FUNCTION_BLOCK "FB24 - Gestione Mov Assi"	// FB 24
TITLE = GESTIONE ASSI STAZIONE OP60
VERSION : 0.1
VAR_INPUT
  INDIRIZZO_INIZIALE_E_A : DINT ;	//INDIRIZZO INIZIALE I/O (VEDI CONFIGURAZIONE HARDWARE)
  OK_FOR_COMMANDS : BOOL ;	//TUTTO PRONTO PER I COMANDI
  RESET_ALLARMI : BOOL ;	//1=RESET ALLARMI AZIONAMENTO
  STOP : BOOL ;	//0=STOP DI TUTTI I MOVIMENTI
  TARGET_POSIZIONE : DINT ;	//TARGET DI POSIZIONAMENTO ASSOLUTO
  TARGET_INCREMENTALE : DINT ;	//SPOSTAMENTO IN MODO INCREMENTALE
  OVERRIDE : INT ;	//OVVERIDE DI VELOCITA'
  JOG_PIU : BOOL ;	//COMANDO JOG PIU'
  JOG_MENO : BOOL ;	//COMANDO JOG MENO
  IN_PKE : WORD ;
  IN_IND : WORD ;
  IN_PWE : DINT ;
  ASSE_SU_HOME : BOOL ;	//ASSE GIA' SU POSIZIONE DI HOME
END_VAR
VAR_OUTPUT
  OUT_PKE : WORD ;
  OUT_IND : WORD ;
  OUT_PWE : DINT ;
  POSIZIONE_ATTUALE : DINT ;
  POSIZIONE_RAGGIUNTA : BOOL ;	//POSIZIONAMENTO ULTIMATO
  HOME_OK : BOOL ;	//1=ASSE RIFERITO
  RIPOSIZIONAMENTO_OK : BOOL ;	//1=RIPOSIZIONAMENTO EFFETTUATO
  ASSE_FERMO_NO_JOB : BOOL ;	//1=ASSE FERMO E NESSUN JOB IN CORSO
  AZIONAMENTO_OK : BOOL ;	//1=AZIONAMENTO PRONTO
  AZIONAMENTO_FAULT : BOOL ;	//1=AZIONAMENTO IN ALLARME
  CAMMA_DI_RIFERIMENTO : BOOL ;	//1=ASSE SU CAMMA DI RIFERIMENTO
  OLTRECORSA_NEGATIVO : BOOL ;	//1=ASSE SU OLTRECORSA HARDWARE NEGATIVO
  OLTRECORSA_POSITIVO : BOOL ;	//1=ASSE SU OLTRECORSA HARDWARE POSITIVO
  FINECORSA_SOFTWARE_NEG : BOOL ;	//1=FINECORSA SOFTWARE NEGATIVO
  FINECORSA_SOFTWARE_POS : BOOL ;	//1=FINECORSA SOFTWARE POSITIVO
  FRENO : BOOL ;	//1=APRIRE IL FRENO DI STAZIONAMENTO
END_VAR
VAR_IN_OUT
  START_ASSOLUTO : BOOL ;	//1=START POSIZIONAMENTO ASSOLUTO
  START_INCREMENTALE : BOOL ;	//1=START POSIZIONAMENTO INCREMENTALE
  START_HOME : BOOL ;	//1=START RICERCA ZERO
  START_RIPOSIZIONAMENTO : BOOL ;	//1=START POSIZIONAMENTO SU POSIZIONE INIZIALE
END_VAR
VAR
  SCELTA_BLOCCO : WORD ;
  BLOCCO_ATTUALE : WORD ;
  INVIA_JOB1 : BOOL ;	//INVIO COMANDO DI CARICA BLOCCO ASSOLUTO
  JOB1_ULTIMATO : BOOL ;	//IL NUOVO BLOCCO DI MOVIMENTO ASSOLUTO E' STATO INVIATO
  INVIA_JOB2 : BOOL ;	//INVIO COMANDO DI CARICA BLOCCO INCREMENTALE
  JOB2_ULTIMATO : BOOL ;	//IL NUOVO BLOCCO DI MOVIMENTO INCREMENTALE E' STATO INVIATO
  GIA_IN_POSIZIONE : BOOL ;	//POSIZIONAMENTO NON NECESSARIO PER ASSE GIA' IN POSIZIONE
  PACO1 : STRUCT
   PACO1_8 : BOOL ;	//1=MARCIA A IMPULSI 1
   PACO1_9 : BOOL ;	//1=MARCIA 1 IMPULSI 2
   PACO1_10 : BOOL ;	//1=ABILITA IL COMANDO (DA METTERE A 1 QUANDO PAST1.9=1)
   PACO1_11 : BOOL ;	//1=AVVIA IL RIFERIMENTO DELL'ASSE
   PACO1_12 : BOOL ;	//RISERVATO
   PACO1_13 : BOOL ;	//1=CAMBIO BLOCCO ESTERNO
   PACO1_14 : BOOL ;	//RISERVATO
   PACO1_15 : BOOL ;	//RISERVATO
   PACO1_0 : BOOL ;	//1=INSERITO 0=DISINSERITO
   PACO1_1 : BOOL ;	//1=INSERITO 0=DISINSERITO
   PACO1_2 : BOOL ;	//1=INSERITO 0=DISINSERITO
   PACO1_3 : BOOL ;	//0=BLOCCO IMPULSI (IL MOTORE SI FERMA PER INERZIA)
   PACO1_4 : BOOL ;	//1=OK 0=STOP ASSE E CANCELLAZIONE PERCORSO RESISDUO
   PACO1_5 : BOOL ;	//1=OK 0=STOP ASSE E ULTIMAZIONE MOVIMENTO CON FRONTE 0-->1
   PACO1_6 : BOOL ;	//0-->1=ATTIVARE L'ORDINE DI SPOSTAMENTO
   PACO1_7 : BOOL ;	//1=TACITAZIONE ALLARME
  END_STRUCT ;
  PAST1 : STRUCT
   PAST1_8 : BOOL ;	//1=NESSUN ERRORE D'INSEGUIMENTO
   PAST1_9 : BOOL ;	//1=SLAVE OK E PRONTO A RICEVERE COMANDI
   PAST1_10 : BOOL ;	//1=POSIZIONE RAGGIUNTA
   PAST1_11 : BOOL ;	//1=ASSE RIFERITO
   PAST1_12 : BOOL ;	//1=POSIZIONAMENTO IN CORSO
   PAST1_13 : BOOL ;	//1=MOTORE FERMO
   PAST1_14 : BOOL ;	//RISERVATO
   PAST1_15 : BOOL ;	//RISERVATO
   PAST1_0 : BOOL ;	//1=PRONTO ALL'INSERZIONE
   PAST1_1 : BOOL ;	//1=PRONTO AL FUNZIONAMENTO
   PAST1_2 : BOOL ;	//STATO ABILITAZIONE REGOLATORE
   PAST1_3 : BOOL ;	//1=PRESEZA GUASTI
   PAST1_4 : BOOL ;	//1=DISINSERIMENTO 2 ASSENTE
   PAST1_5 : BOOL ;	//1=DISINSERIMENTO 3 ASSENTE
   PAST1_6 : BOOL ;	//1=BLOCCO ALL'INSERZIONE
   PAST1_7 : BOOL ;	//1=PRESENZA AVVISI
  END_STRUCT ;
  DIGin : STRUCT
   DIGin_8 : BOOL ;
   DIGin_9 : BOOL ;
   DIGin_10 : BOOL ;
   DIGin_11 : BOOL ;
   DIGin_12 : BOOL ;
   DIGin_13 : BOOL ;
   DIGin_14 : BOOL ;
   DIGin_15 : BOOL ;
   DIGin_0 : BOOL ;	//1=ASSE SU CAMMA DI HOME
   DIGin_1 : BOOL ;	//1=ASSE SU EXTRACORSA NEGATIVO
   DIGin_2 : BOOL ;	//1=ASSE SU EXTRACORSA POSITIVO
   DIGin_3 : BOOL ;
   DIGin_4 : BOOL ;
   DIGin_5 : BOOL ;
   DIGin_6 : BOOL ;
   DIGin_7 : BOOL ;
  END_STRUCT ;
  AUX1 : BOOL ;	//APPOGGIO PER FRONTE
  AUX2 : BOOL ;	//APPOGGIO PER FRONTE
  AUX3 : BOOL ;	//APPOGGIO PER FRONTE
  AUX4 : BOOL ;	//APPOGGIO PER FRONTE
  AUX5 : BOOL ;	//APPOGGIO PER FRONTE
  AUX6 : BOOL ;	//APPOGGIO PER FRONTE
  AUX7 : BOOL ;	//APPOGGIO PER FRONTE
  VERIFICA_SPOSTAMENTO : DINT ;	//DIFFERENZA TRA TARGET E POSIZIONE ATTUALE
  PAST2 : STRUCT
   PAST2_8 : BOOL ;	//1=TACITARE IL GUASTO 608
   PAST2_9 : BOOL ;	//1=ATTUALE MOTORE 1.SEGNALE
   PAST2_10 : BOOL ;	//1=ATTUALE MOTORE 2.SEGNALE
   PAST2_11 : BOOL ;	//1=RISERVATO
   PAST2_12 : BOOL ;
   PAST2_13 : BOOL ;
   PAST2_14 : BOOL ;
   PAST2_15 : BOOL ;
   PAST2_0 : BOOL ;
   PAST2_1 : BOOL ;
   PAST2_2 : BOOL ;
   PAST2_3 : BOOL ;	//PRIMO FILTRO DEL RIFERIMENTO ATTIVO
   PAST2_4 : BOOL ;	//BLOCCO DELL'INTEGRATORE NEL REGOLATORE DI VELOCITA'
   PAST2_5 : BOOL ;	//APRIRE IL FRENO DI STAZIONAMENTO
   PAST2_6 : BOOL ;	//BLOCCO DELL'INTEGRATORE NEL REGOLATORE DI VELOCITA'
   PAST2_7 : BOOL ;	//SCELTO L'ASSE IN PARCHEGGIO
  END_STRUCT ;
  POS_PAST : STRUCT
   POS_PAST_0 : BOOL ;	//FUNZIONAMENTO A SEGUIRE
   POS_PAST_1 : BOOL ;	//LIMITAZIONE DELLA VELOCITA' LINEARE ATTIVA
   POS_PAST_2 : BOOL ;	//C'E' IL RIFERIMENTO
   POS_PAST_3 : BOOL ;	//BIT DI FUNZIONE
   POS_PAST_4 : BOOL ;	//L'ASSE SI SPOSTA IN AVANTI
   POS_PAST_5 : BOOL ;	//L'ASSE SI SPOSTA INDIETRO
   POS_PAST_6 : BOOL ;	//FINECORSA SOFTWARE MENO
   POS_PAST_7 : BOOL ;	//FINECORSA SOFTWARE PIU'
   POS_PAST_8 : BOOL ;	//SEGNALE D'INSERZIONE DELLA CAMMA 1
   POS_PAST_9 : BOOL ;	//SEGNALE D'INSERZIONE DELLA CAMMA 2
   POS_PAST_10 : BOOL ;	//USCITA DIRETTA 1 CON IL BLOCCO DI SPOSTAMENTO
   POS_PAST_11 : BOOL ;	//USCITA DIRETTA 2 CON IL BLOCCO DI SPOSTAMENTO
   POS_PAST_12 : BOOL ;	//RISERVATO
   POS_PAST_13 : BOOL ;	//RISERVATO
   POS_PAST_14 : BOOL ;	//RISERVATO
   POS_PAST_15 : BOOL ;	//RISERVATO
  END_STRUCT ;
END_VAR
BEGIN
NETWORK
TITLE = AGGIORNAMENTO IMMAGINE INGRESSI
      L     #INDIRIZZO_INIZIALE_E_A;
      L     8;
      +I;
      SLD   3;
      T     MD 100;
      L     PIW [MD 100];	//;PAST1
      T     DIW 52;
      L     MD 100;
      SRW   3;
      L     2;
      +D;
      SLW   3;
      T     MD 100;
//;
      L     PIW [MD 100];	//;BLOCCO ATTUALE
      T     #BLOCCO_ATTUALE;
      L     MD 100;
      SRW   3;
      L     2;
      +D;
      SLW   3;
      T     MD 100;
//;
      L     PIW [MD 100];	//;POS PAST
      T     DIW 64;
      L     MD 100;
      SRW   3;
      L     2;
      +D;
      SLW   3;
      T     MD 100;
//;
      L     PIW [MD 100];	//;PAST 2
      T     DIW 62;
      L     MD 100;
      SRW   3;
      L     2;
      +D;
      SLW   3;
      T     MD 100;
//;
      L     PID [MD 100];	//; POSIZIONE ATTUALE
      T     #POSIZIONE_ATTUALE;
      L     MD 100;
      SRW   3;
      L     4;
      +D;
      SLW   3;
      T     MD 100;
//;
      L     PIW [MD 100];	//;INGRESSI DIGITALI
      T     DIW 54;
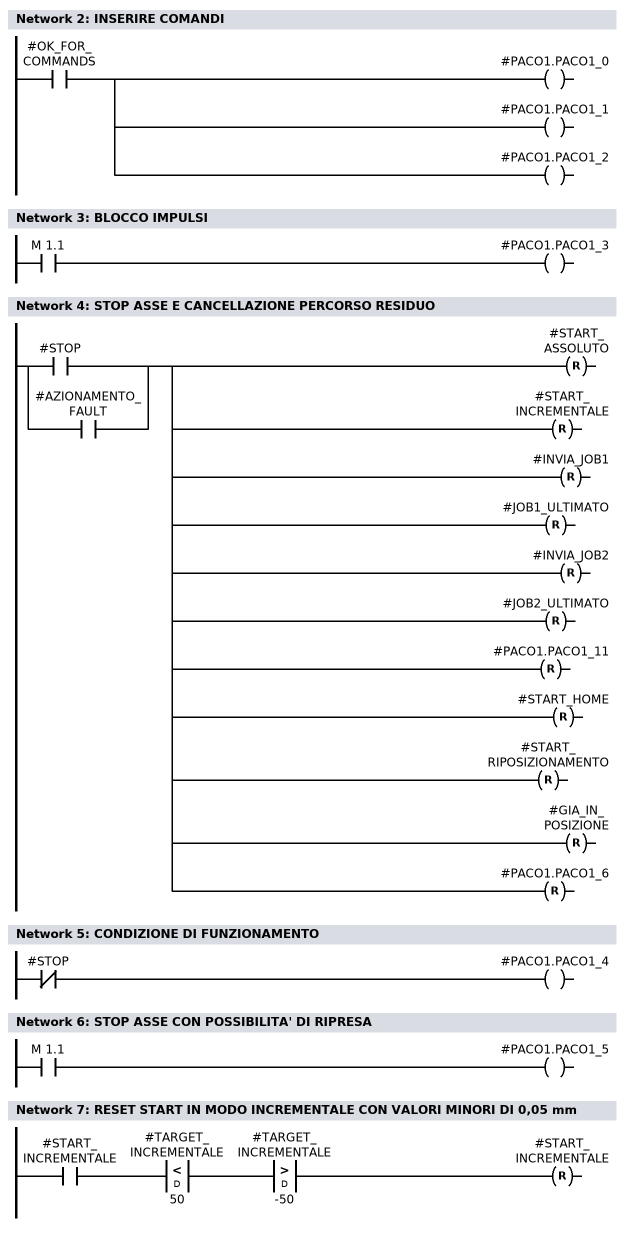
NETWORK
TITLE = INSERIRE COMANDI
      A     #OK_FOR_COMMANDS;
      =     #PACO1.PACO1_0;
      =     #PACO1.PACO1_1;
      =     #PACO1.PACO1_2;
NETWORK
TITLE = BLOCCO IMPULSI
      A     M 1.1;
      =     #PACO1.PACO1_3;
NETWORK
TITLE = STOP ASSE E CANCELLAZIONE PERCORSO RESIDUO
      O     #STOP;
      O     #AZIONAMENTO_FAULT;
      R     #START_ASSOLUTO;
      R     #START_INCREMENTALE;
      R     #INVIA_JOB1;
      R     #JOB1_ULTIMATO;
      R     #INVIA_JOB2;
      R     #JOB2_ULTIMATO;
      R     #PACO1.PACO1_11;
      R     #START_HOME;
      R     #START_RIPOSIZIONAMENTO;
      R     #GIA_IN_POSIZIONE;
      R     #PACO1.PACO1_6;
NETWORK
TITLE = CONDIZIONE DI FUNZIONAMENTO
      AN    #STOP;
      =     #PACO1.PACO1_4;
NETWORK
TITLE = STOP ASSE CON POSSIBILITA' DI RIPRESA 
      A     M 1.1;
      =     #PACO1.PACO1_5;
NETWORK
TITLE = RESET START IN MODO INCREMENTALE CON VALORI MINORI DI 0,05 mm
      A     #START_INCREMENTALE;
      A(;
      L     #TARGET_INCREMENTALE;
      L     50;
      <D;
      );
      A(;
      L     #TARGET_INCREMENTALE;
      L     -50;
      >D;
      );
      R     #START_INCREMENTALE;
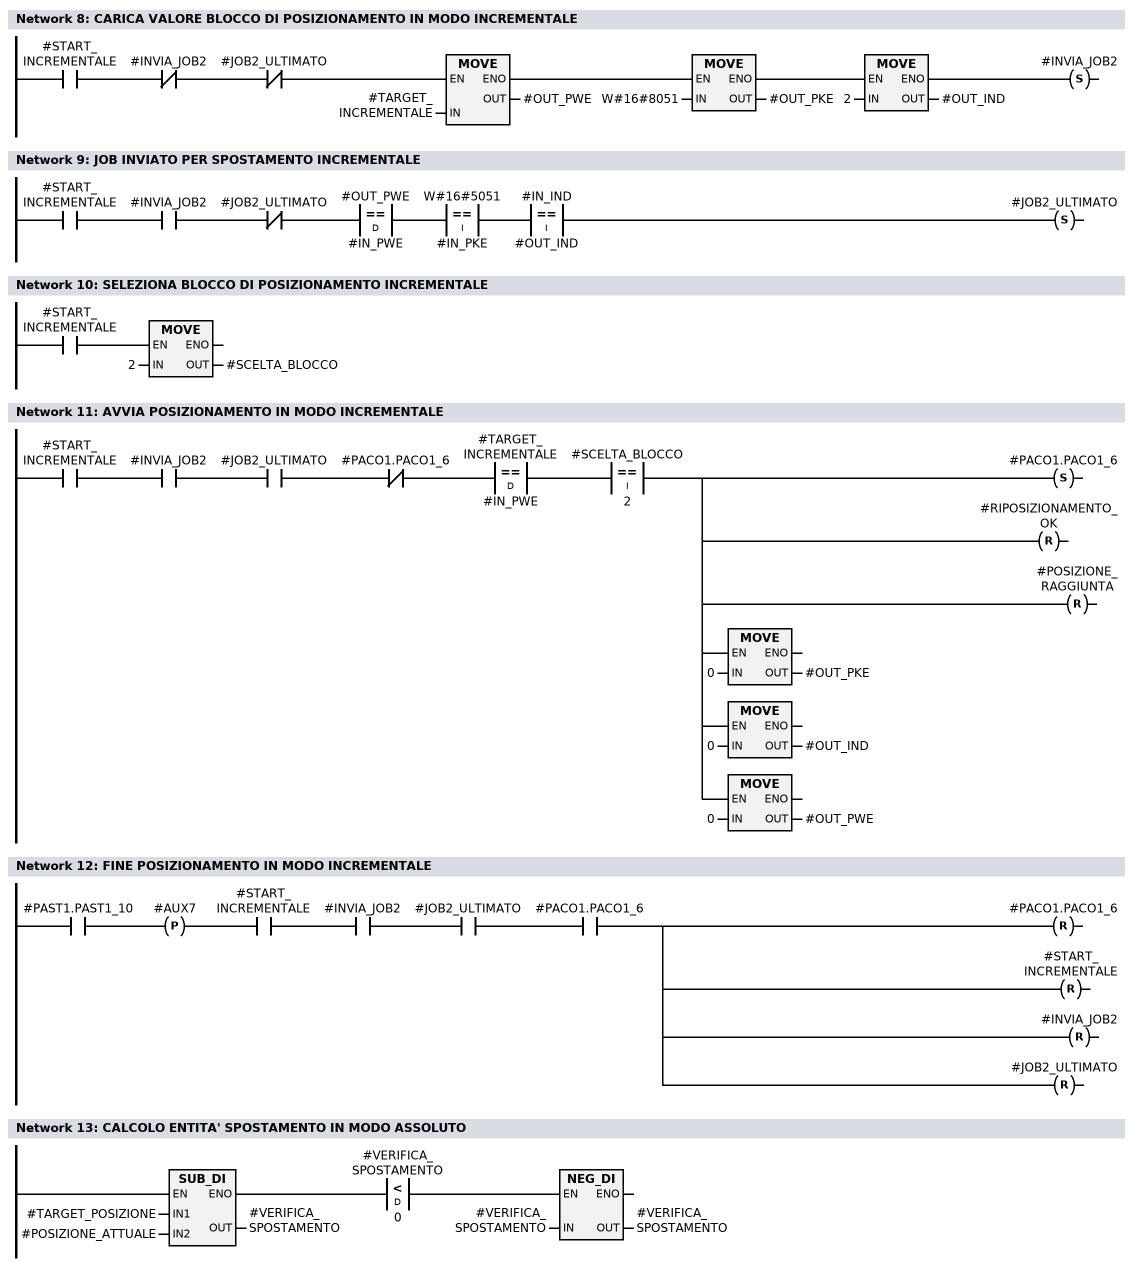
NETWORK
TITLE = CARICA VALORE BLOCCO DI POSIZIONAMENTO IN MODO INCREMENTALE
      A(;
      A(;
      A     #START_INCREMENTALE;
      AN    #INVIA_JOB2;
      AN    #JOB2_ULTIMATO;
      JNB   _001;
      L     #TARGET_INCREMENTALE;
      T     #OUT_PWE;
      SET;
      SAVE;
      CLR;
_001: A     BR;
      );
      JNB   _002;
      L     W#16#8051;
      T     #OUT_PKE;
      SET;
      SAVE;
      CLR;
_002: A     BR;
      );
      JNB   _003;
      L     2;
      T     #OUT_IND;
      SET;
      SAVE;
      CLR;
_003: A     BR;
      S     #INVIA_JOB2;
NETWORK
TITLE = JOB INVIATO PER SPOSTAMENTO INCREMENTALE
      A     #START_INCREMENTALE;
      A     #INVIA_JOB2;
      AN    #JOB2_ULTIMATO;
      A(;
      L     #OUT_PWE;
      L     #IN_PWE;
      ==D;
      );
      A(;
      L     W#16#5051;
      L     #IN_PKE;
      ==I;
      );
      A(;
      L     #IN_IND;
      L     #OUT_IND;
      ==I;
      );
      S     #JOB2_ULTIMATO;
NETWORK
TITLE = SELEZIONA BLOCCO DI POSIZIONAMENTO INCREMENTALE
      A     #START_INCREMENTALE;
      JNB   _004;
      L     2;
      T     #SCELTA_BLOCCO;
_004: NOP   0;
NETWORK
TITLE = AVVIA POSIZIONAMENTO IN MODO INCREMENTALE
      A     #START_INCREMENTALE;
      A     #INVIA_JOB2;
      A     #JOB2_ULTIMATO;
      AN    #PACO1.PACO1_6;
      A(;
      L     #TARGET_INCREMENTALE;
      L     #IN_PWE;
      ==D;
      );
      A(;
      L     #SCELTA_BLOCCO;
      L     2;
      ==I;
      );
      =     L 0.0;
      A     L 0.0;
      BLD   102;
      S     #PACO1.PACO1_6;
      A     L 0.0;
      BLD   102;
      R     #RIPOSIZIONAMENTO_OK;
      A     L 0.0;
      BLD   102;
      R     #POSIZIONE_RAGGIUNTA;
      A     L 0.0;
      JNB   _005;
      L     0;
      T     #OUT_PKE;
_005: NOP   0;
      A     L 0.0;
      JNB   _006;
      L     0;
      T     #OUT_IND;
_006: NOP   0;
      A     L 0.0;
      JNB   _007;
      L     0;
      T     #OUT_PWE;
_007: NOP   0;
NETWORK
TITLE = FINE POSIZIONAMENTO IN MODO INCREMENTALE
      A     #PAST1.PAST1_10;
      FP    #AUX7;
      A     #START_INCREMENTALE;
      A     #INVIA_JOB2;
      A     #JOB2_ULTIMATO;
      A     #PACO1.PACO1_6;
      R     #PACO1.PACO1_6;
      R     #START_INCREMENTALE;
      R     #INVIA_JOB2;
      R     #JOB2_ULTIMATO;
NETWORK
TITLE = CALCOLO ENTITA' SPOSTAMENTO IN MODO ASSOLUTO
      A(;
      L     #TARGET_POSIZIONE;
      L     #POSIZIONE_ATTUALE;
      -D;
      T     #VERIFICA_SPOSTAMENTO;
      AN    OV;
      SAVE;
      CLR;
      A     BR;
      );
      A(;
      L     #VERIFICA_SPOSTAMENTO;
      L     0;
      <D;
      );
      JNB   _008;
      L     #VERIFICA_SPOSTAMENTO;
      NEGD;
      T     #VERIFICA_SPOSTAMENTO;
_008: NOP   0;
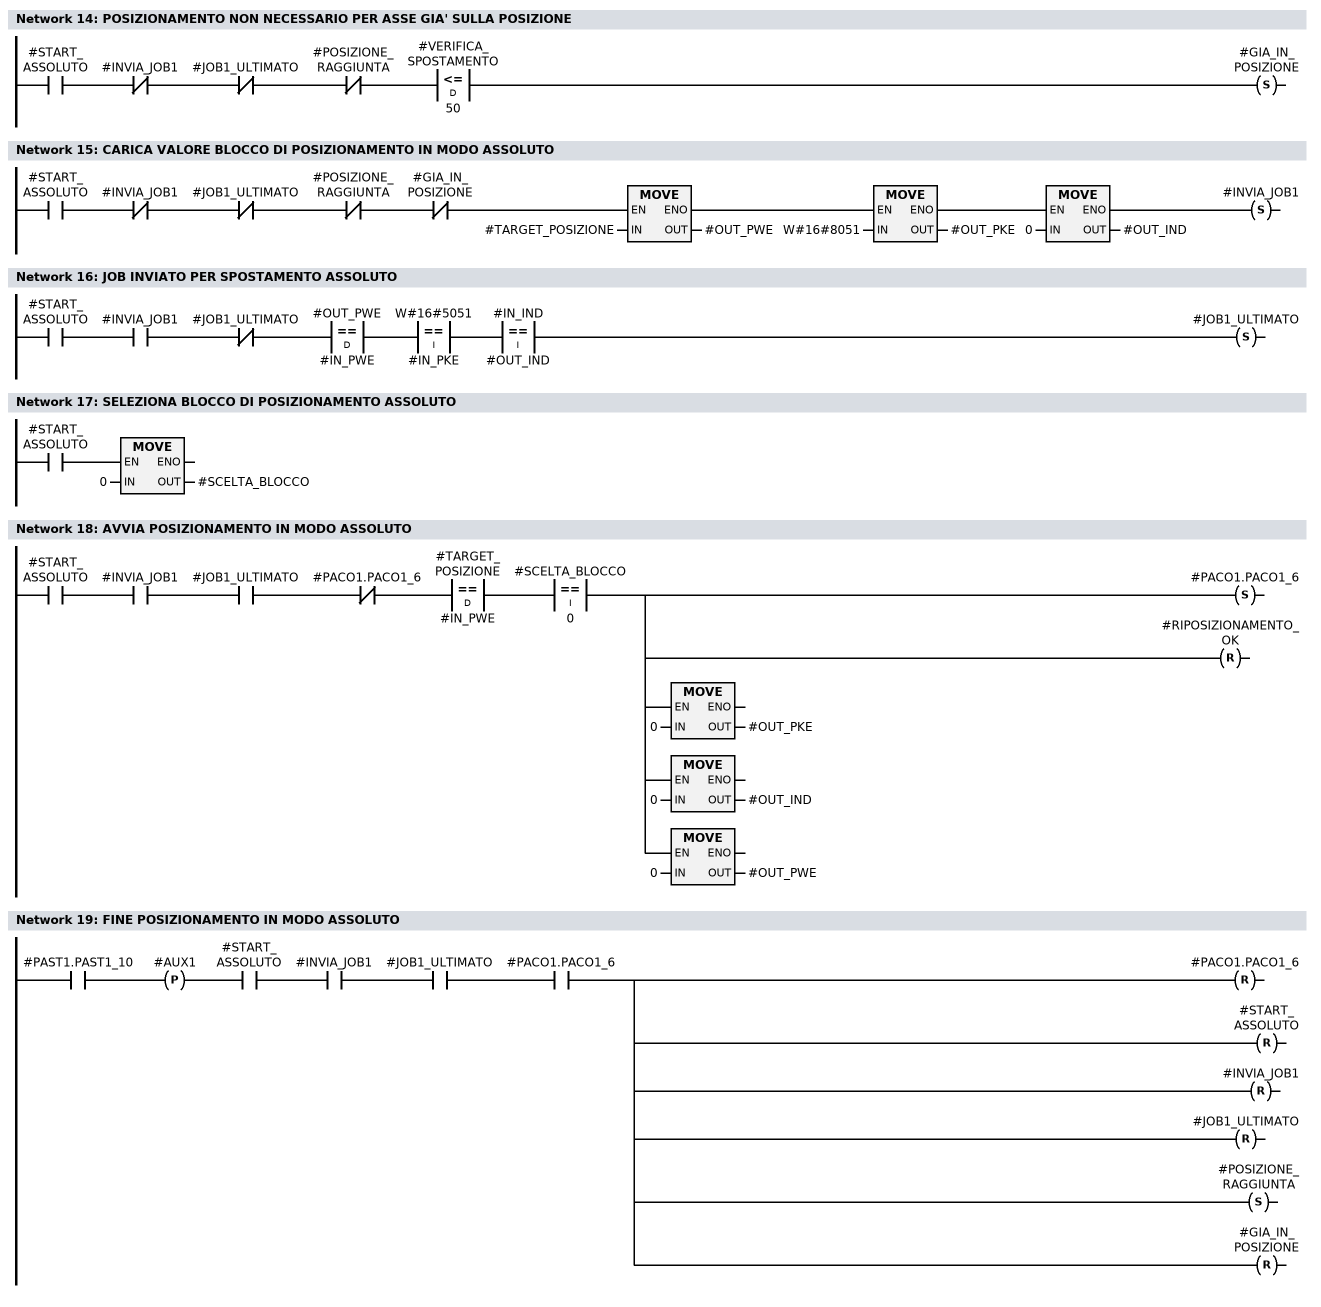
NETWORK
TITLE = POSIZIONAMENTO NON NECESSARIO PER ASSE GIA' SULLA POSIZIONE
      A     #START_ASSOLUTO;
      AN    #INVIA_JOB1;
      AN    #JOB1_ULTIMATO;
      AN    #POSIZIONE_RAGGIUNTA;
      A(;
      L     #VERIFICA_SPOSTAMENTO;
      L     50;
      <=D;
      );
      S     #GIA_IN_POSIZIONE;
NETWORK
TITLE = CARICA VALORE BLOCCO DI POSIZIONAMENTO IN MODO ASSOLUTO
      A(;
      A(;
      A     #START_ASSOLUTO;
      AN    #INVIA_JOB1;
      AN    #JOB1_ULTIMATO;
      AN    #POSIZIONE_RAGGIUNTA;
      AN    #GIA_IN_POSIZIONE;
      JNB   _009;
      L     #TARGET_POSIZIONE;
      T     #OUT_PWE;
      SET;
      SAVE;
      CLR;
_009: A     BR;
      );
      JNB   _00a;
      L     W#16#8051;
      T     #OUT_PKE;
      SET;
      SAVE;
      CLR;
_00a: A     BR;
      );
      JNB   _00b;
      L     0;
      T     #OUT_IND;
      SET;
      SAVE;
      CLR;
_00b: A     BR;
      S     #INVIA_JOB1;
NETWORK
TITLE = JOB INVIATO PER SPOSTAMENTO ASSOLUTO
      A     #START_ASSOLUTO;
      A     #INVIA_JOB1;
      AN    #JOB1_ULTIMATO;
      A(;
      L     #OUT_PWE;
      L     #IN_PWE;
      ==D;
      );
      A(;
      L     W#16#5051;
      L     #IN_PKE;
      ==I;
      );
      A(;
      L     #IN_IND;
      L     #OUT_IND;
      ==I;
      );
      S     #JOB1_ULTIMATO;
NETWORK
TITLE = SELEZIONA BLOCCO DI POSIZIONAMENTO ASSOLUTO
      A     #START_ASSOLUTO;
      JNB   _00c;
      L     0;
      T     #SCELTA_BLOCCO;
_00c: NOP   0;
NETWORK
TITLE = AVVIA POSIZIONAMENTO IN MODO ASSOLUTO
      A     #START_ASSOLUTO;
      A     #INVIA_JOB1;
      A     #JOB1_ULTIMATO;
      AN    #PACO1.PACO1_6;
      A(;
      L     #TARGET_POSIZIONE;
      L     #IN_PWE;
      ==D;
      );
      A(;
      L     #SCELTA_BLOCCO;
      L     0;
      ==I;
      );
      =     L 0.0;
      A     L 0.0;
      BLD   102;
      S     #PACO1.PACO1_6;
      A     L 0.0;
      BLD   102;
      R     #RIPOSIZIONAMENTO_OK;
      A     L 0.0;
      JNB   _00d;
      L     0;
      T     #OUT_PKE;
_00d: NOP   0;
      A     L 0.0;
      JNB   _00e;
      L     0;
      T     #OUT_IND;
_00e: NOP   0;
      A     L 0.0;
      JNB   _00f;
      L     0;
      T     #OUT_PWE;
_00f: NOP   0;
NETWORK
TITLE = FINE POSIZIONAMENTO IN MODO ASSOLUTO
      A     #PAST1.PAST1_10;
      FP    #AUX1;
      A     #START_ASSOLUTO;
      A     #INVIA_JOB1;
      A     #JOB1_ULTIMATO;
      A     #PACO1.PACO1_6;
      R     #PACO1.PACO1_6;
      R     #START_ASSOLUTO;
      R     #INVIA_JOB1;
      R     #JOB1_ULTIMATO;
      S     #POSIZIONE_RAGGIUNTA;
      R     #GIA_IN_POSIZIONE;
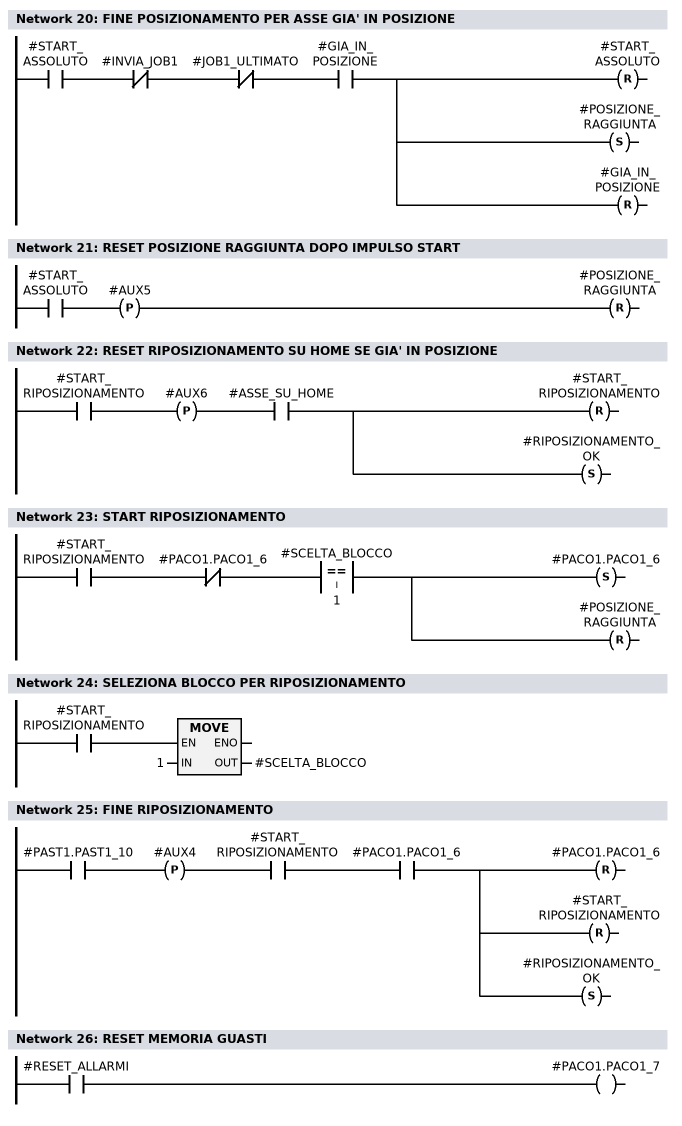
NETWORK
TITLE = FINE POSIZIONAMENTO PER ASSE GIA' IN POSIZIONE
      A     #START_ASSOLUTO;
      AN    #INVIA_JOB1;
      AN    #JOB1_ULTIMATO;
      A     #GIA_IN_POSIZIONE;
      R     #START_ASSOLUTO;
      S     #POSIZIONE_RAGGIUNTA;
      R     #GIA_IN_POSIZIONE;
NETWORK
TITLE = RESET POSIZIONE RAGGIUNTA DOPO IMPULSO START
      A     #START_ASSOLUTO;
      FP    #AUX5;
      R     #POSIZIONE_RAGGIUNTA;
NETWORK
TITLE = RESET RIPOSIZIONAMENTO SU HOME SE GIA' IN POSIZIONE
      A     #START_RIPOSIZIONAMENTO;
      FP    #AUX6;
      A     #ASSE_SU_HOME;
      R     #START_RIPOSIZIONAMENTO;
      S     #RIPOSIZIONAMENTO_OK;
NETWORK
TITLE = START RIPOSIZIONAMENTO
      A     #START_RIPOSIZIONAMENTO;
      AN    #PACO1.PACO1_6;
      A(;
      L     #SCELTA_BLOCCO;
      L     1;
      ==I;
      );
      S     #PACO1.PACO1_6;
      R     #POSIZIONE_RAGGIUNTA;
NETWORK
TITLE = SELEZIONA BLOCCO PER RIPOSIZIONAMENTO
      A     #START_RIPOSIZIONAMENTO;
      JNB   _010;
      L     1;
      T     #SCELTA_BLOCCO;
_010: NOP   0;
NETWORK
TITLE = FINE RIPOSIZIONAMENTO
      A     #PAST1.PAST1_10;
      FP    #AUX4;
      A     #START_RIPOSIZIONAMENTO;
      A     #PACO1.PACO1_6;
      R     #PACO1.PACO1_6;
      R     #START_RIPOSIZIONAMENTO;
      S     #RIPOSIZIONAMENTO_OK;
NETWORK
TITLE = RESET MEMORIA GUASTI
      A     #RESET_ALLARMI;
      =     #PACO1.PACO1_7;
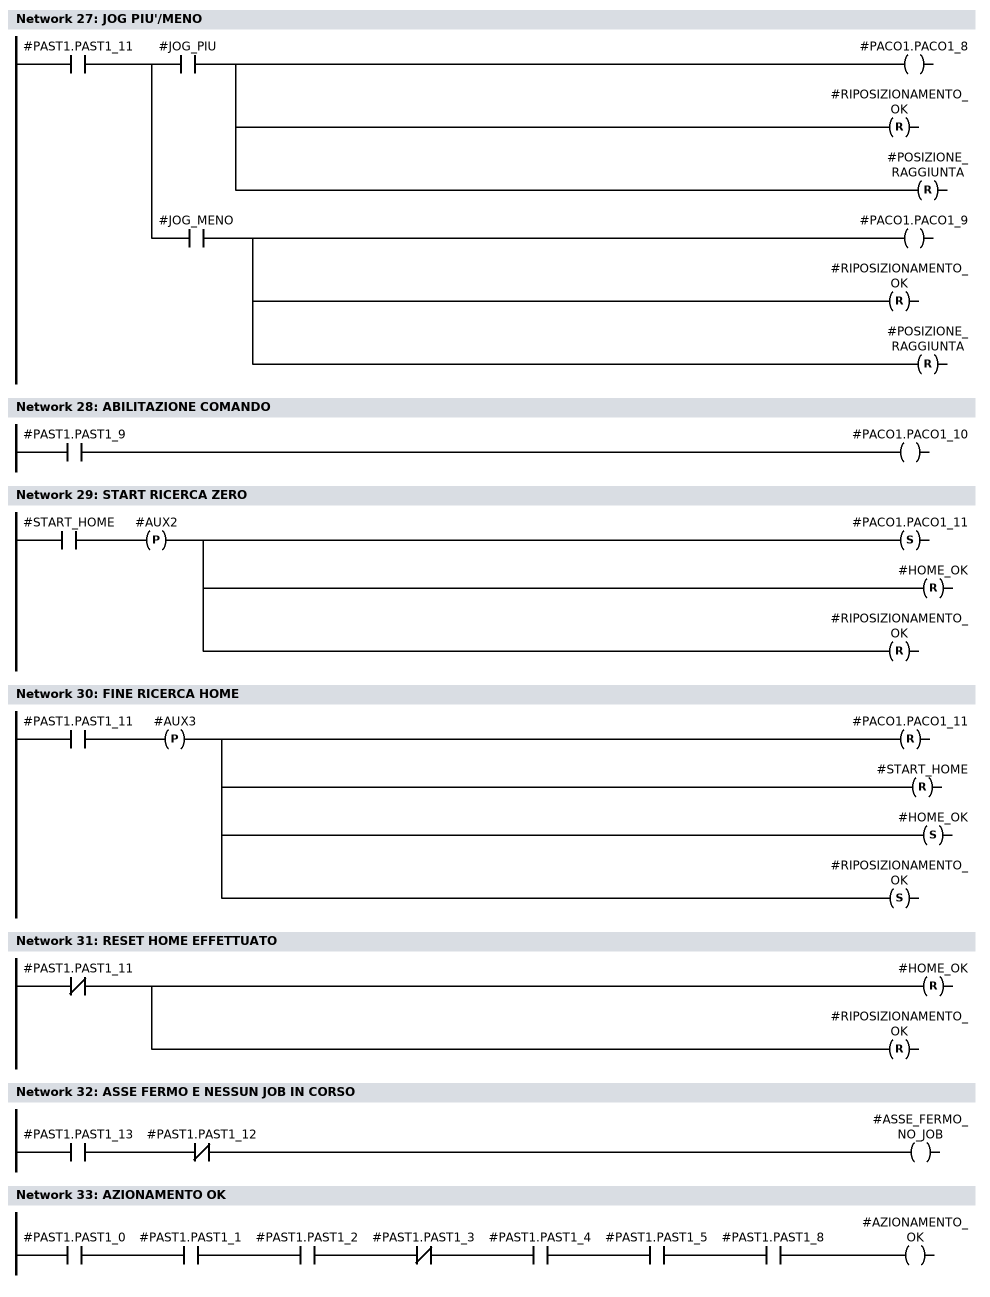
NETWORK
TITLE = JOG PIU'/MENO
      A     #PAST1.PAST1_11;
      =     L 0.0;
      A     L 0.0;
      A     #JOG_PIU;
      =     #PACO1.PACO1_8;
      R     #RIPOSIZIONAMENTO_OK;
      R     #POSIZIONE_RAGGIUNTA;
      A     L 0.0;
      A     #JOG_MENO;
      =     #PACO1.PACO1_9;
      R     #RIPOSIZIONAMENTO_OK;
      R     #POSIZIONE_RAGGIUNTA;
NETWORK
TITLE = ABILITAZIONE COMANDO
      A     #PAST1.PAST1_9;
      =     #PACO1.PACO1_10;
NETWORK
TITLE = START RICERCA ZERO
      A     #START_HOME;
      FP    #AUX2;
      S     #PACO1.PACO1_11;
      R     #HOME_OK;
      R     #RIPOSIZIONAMENTO_OK;
NETWORK
TITLE = FINE RICERCA HOME
      A     #PAST1.PAST1_11;
      FP    #AUX3;
      R     #PACO1.PACO1_11;
      R     #START_HOME;
      S     #HOME_OK;
      S     #RIPOSIZIONAMENTO_OK;
NETWORK
TITLE = RESET HOME EFFETTUATO
      AN    #PAST1.PAST1_11;
      R     #HOME_OK;
      R     #RIPOSIZIONAMENTO_OK;
NETWORK
TITLE = ASSE FERMO E NESSUN JOB IN CORSO
      A     #PAST1.PAST1_13;
      AN    #PAST1.PAST1_12;
      =     #ASSE_FERMO_NO_JOB;
NETWORK
TITLE = AZIONAMENTO OK
      A     #PAST1.PAST1_0;
      A     #PAST1.PAST1_1;
      A     #PAST1.PAST1_2;
      AN    #PAST1.PAST1_3;
      A     #PAST1.PAST1_4;
      A     #PAST1.PAST1_5;
      A     #PAST1.PAST1_8;
      =     #AZIONAMENTO_OK;
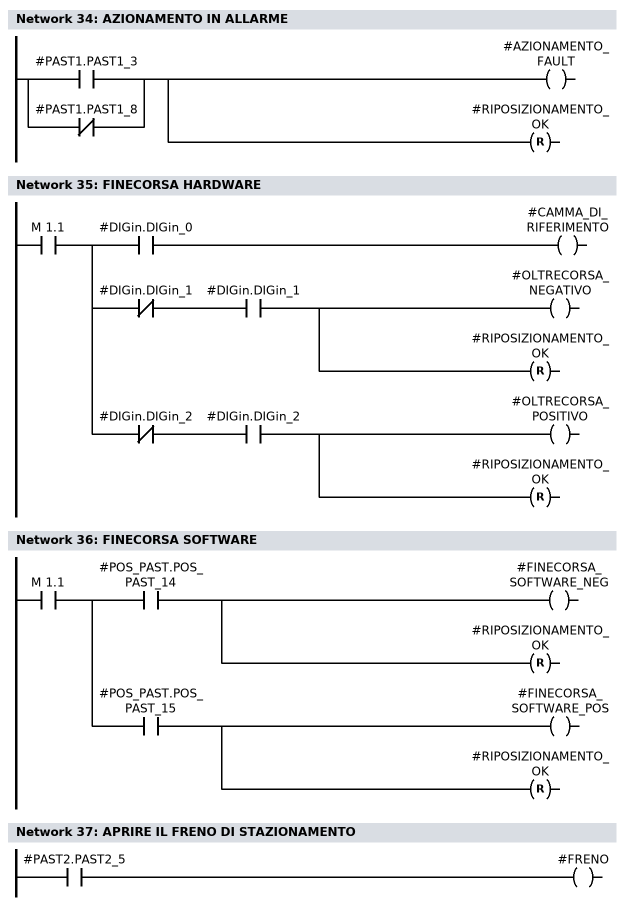
NETWORK
TITLE = AZIONAMENTO IN ALLARME
      O     #PAST1.PAST1_3;
      ON    #PAST1.PAST1_8;
      =     #AZIONAMENTO_FAULT;
      R     #RIPOSIZIONAMENTO_OK;
NETWORK
TITLE = FINECORSA HARDWARE
      A     M 1.1;
      =     L 0.0;
      A     L 0.0;
      A     #DIGin.DIGin_0;
      =     #CAMMA_DI_RIFERIMENTO;
      A     L 0.0;
      AN    #DIGin.DIGin_1;
      A     #DIGin.DIGin_1;
      =     #OLTRECORSA_NEGATIVO;
      R     #RIPOSIZIONAMENTO_OK;
      A     L 0.0;
      AN    #DIGin.DIGin_2;
      A     #DIGin.DIGin_2;
      =     #OLTRECORSA_POSITIVO;
      R     #RIPOSIZIONAMENTO_OK;
NETWORK
TITLE = FINECORSA SOFTWARE
      A     M 1.1;
      =     L 0.0;
      A     L 0.0;
      A     #POS_PAST.POS_PAST_14;
      =     #FINECORSA_SOFTWARE_NEG;
      R     #RIPOSIZIONAMENTO_OK;
      A     L 0.0;
      A     #POS_PAST.POS_PAST_15;
      =     #FINECORSA_SOFTWARE_POS;
      R     #RIPOSIZIONAMENTO_OK;
NETWORK
TITLE = APRIRE IL FRENO DI STAZIONAMENTO
      A     #PAST2.PAST2_5;
      =     #FRENO;
NETWORK
TITLE = AGGIORNAMENTO IMMAGINE USCITE
      L     #INDIRIZZO_INIZIALE_E_A;
      L     8;
      +I;
      SLD   3;
      T     MD 100;
      L     DIW 50;
      T     PQW [MD 100];	//;PACO 1
      L     MD 100;
      SRW   3;
      L     2;
      +D;
      SLW   3;
      T     MD 100;
//;
      L     #SCELTA_BLOCCO;
      T     PQW [MD 100];	//;SCELTA BLOCCO
      L     MD 100;
      SRW   3;
      L     6;
      +D;
      SLW   3;
      T     MD 100;
//;
      L     #OVERRIDE;
      T     PQW [MD 100];	//;OVERRIDE
END_FUNCTION_BLOCK

// FC 7: know-how protected block, not included

FUNCTION "FC11 - STATUS" : VOID	// FC 11
TITLE = Sensors and proximity state
VERSION : 0.1
VAR_TEMP
  temp_INT : INT ;
END_VAR
BEGIN
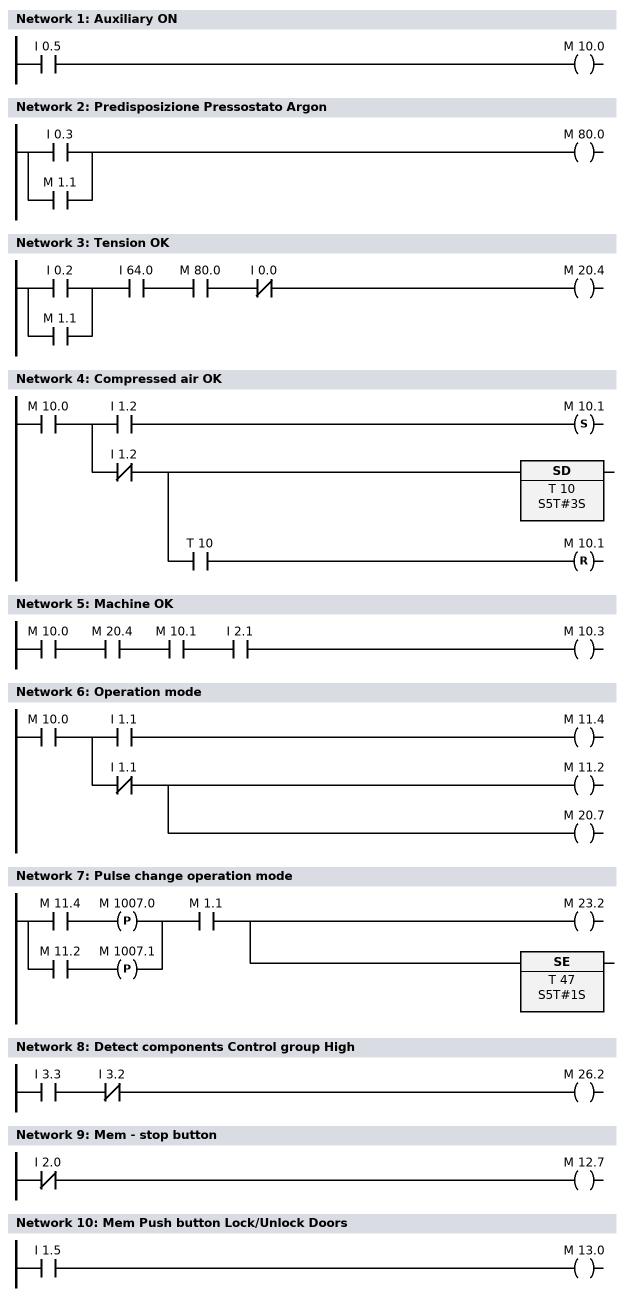
NETWORK
TITLE = Auxiliary ON
      A     I 0.5;
      =     M 10.0;
NETWORK
TITLE = Predisposizione Pressostato Argon
      O     I 0.3;
      O     M 1.1;
      =     M 80.0;
NETWORK
TITLE = Tension OK
      A(;
      O     I 0.2;
      O     M 1.1;
      );
      A     I 64.0;
      A     M 80.0;
      AN    I 0.0;
      =     M 20.4;
NETWORK
TITLE = Compressed air OK
      A     M 10.0;
      =     L 2.0;
      A     L 2.0;
      A     I 1.2;
      S     M 10.1;
      A     L 2.0;
      AN    I 1.2;
      =     L 2.1;
      A     L 2.1;
      BLD   102;
      L     S5T#3S;
      SD    T 10;
      A     L 2.1;
      A     T 10;
      R     M 10.1;
NETWORK
TITLE = Machine OK
      A     M 10.0;
      A     M 20.4;
      A     M 10.1;
      A     I 2.1;
      =     M 10.3;
NETWORK
TITLE = Operation mode
      A     M 10.0;
      =     L 2.0;
      A     L 2.0;
      A     I 1.1;
      =     M 11.4;
      A     L 2.0;
      AN    I 1.1;
      =     M 11.2;
      =     M 20.7;
NETWORK
TITLE = Pulse change operation mode
      A(;
      A     M 11.4;
      FP    M 1007.0;
      O(;
      A     M 11.2;
      FP    M 1007.1;
      );
      );
      A     M 1.1;
      =     M 23.2;
      L     S5T#1S;
      SE    T 47;
NETWORK
TITLE = Detect components Control group High
      A     I 3.3;
      AN    I 3.2;
      =     M 26.2;
NETWORK
TITLE = Mem - stop button
      AN    I 2.0;
      =     M 12.7;
NETWORK
TITLE = Mem Push button Lock/Unlock Doors
      A     I 1.5;
      =     M 13.0;
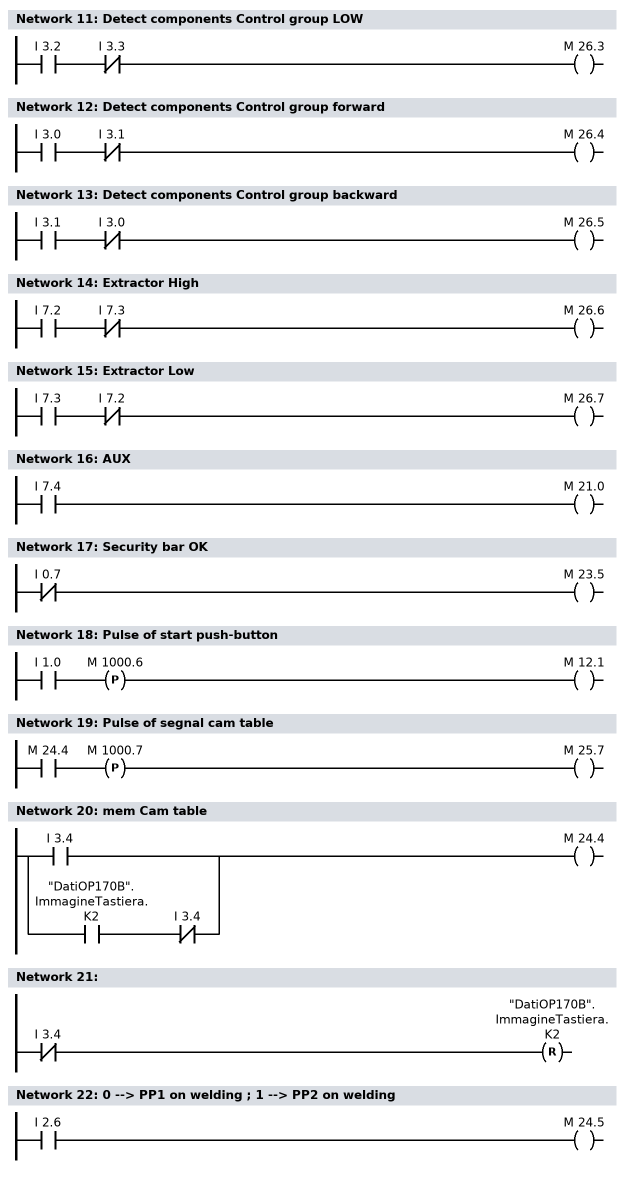
NETWORK
TITLE = Detect components Control group LOW
      A     I 3.2;
      AN    I 3.3;
      =     M 26.3;
NETWORK
TITLE = Detect components Control group forward
      A     I 3.0;
      AN    I 3.1;
      =     M 26.4;
NETWORK
TITLE = Detect components Control group backward
      A     I 3.1;
      AN    I 3.0;
      =     M 26.5;
NETWORK
TITLE = Extractor High
      A     I 7.2;
      AN    I 7.3;
      =     M 26.6;
NETWORK
TITLE = Extractor Low
      A     I 7.3;
      AN    I 7.2;
      =     M 26.7;
NETWORK
TITLE = AUX
      A     I 7.4;
      =     M 21.0;
NETWORK
TITLE = Security bar OK
      AN    I 0.7;
      =     M 23.5;
NETWORK
TITLE = Pulse of start push-button
      A     I 1.0;
      FP    M 1000.6;
      =     M 12.1;
NETWORK
TITLE = Pulse of segnal cam table
      A     M 24.4;
      FP    M 1000.7;
      =     M 25.7;
NETWORK
TITLE = mem Cam table
      O     I 3.4;
      O;
      A     "DatiOP170B".ImmagineTastiera.K2;
      AN    I 3.4;
      =     M 24.4;
NETWORK
TITLE =
      AN    I 3.4;
      R     "DatiOP170B".ImmagineTastiera.K2;
NETWORK
TITLE = 0 --> PP1 on welding ; 1 --> PP2 on welding
      A     I 2.6;
      =     M 24.5;
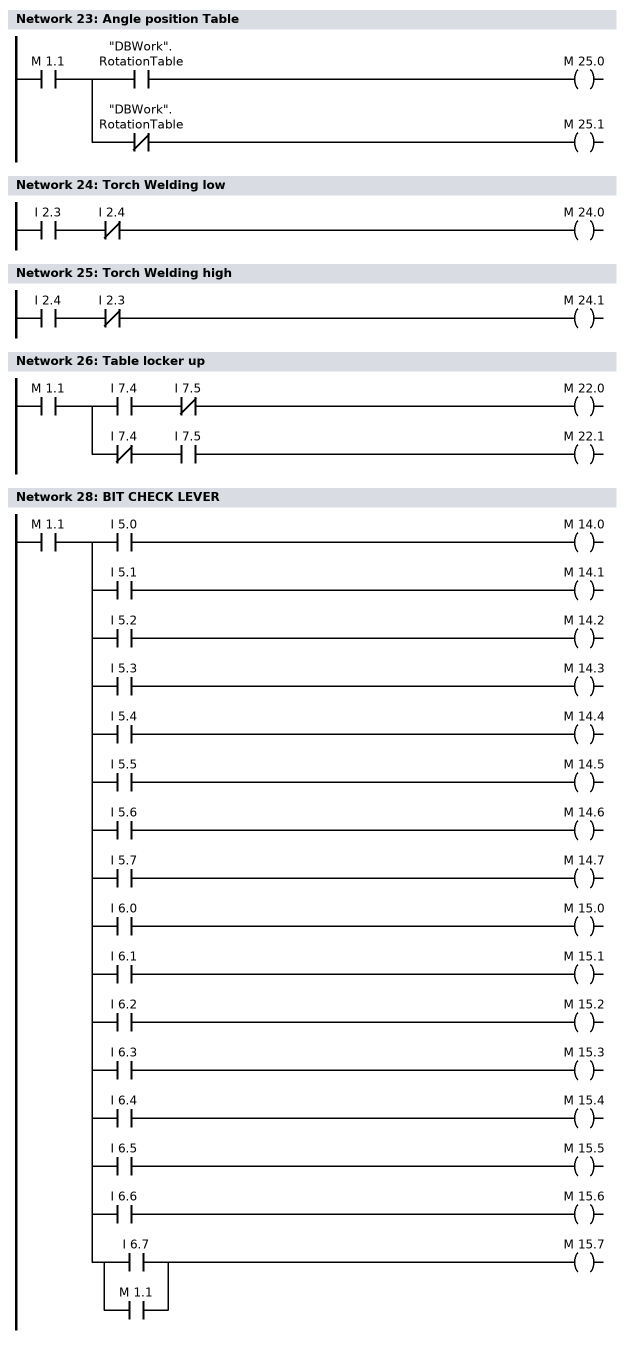
NETWORK
TITLE = Angle position Table
      A     M 1.1;
      =     L 2.0;
      A     L 2.0;
      A     "DBWork".RotationTable;
      =     M 25.0;
      A     L 2.0;
      AN    "DBWork".RotationTable;
      =     M 25.1;
NETWORK
TITLE = Torch Welding low
      A     I 2.3;
      AN    I 2.4;
      =     M 24.0;
NETWORK
TITLE = Torch Welding high
      A     I 2.4;
      AN    I 2.3;
      =     M 24.1;
NETWORK
TITLE = Table locker up
      A     M 1.1;
      =     L 2.0;
      A     L 2.0;
      A     I 7.4;
      AN    I 7.5;
      =     M 22.0;
      A     L 2.0;
      AN    I 7.4;
      A     I 7.5;
      =     M 22.1;
NETWORK
TITLE =
NETWORK
TITLE = BIT CHECK LEVER
      A     M 1.1;
      =     L 2.0;
      A     L 2.0;
      A     I 5.0;
      =     M 14.0;
      A     L 2.0;
      A     I 5.1;
      =     M 14.1;
      A     L 2.0;
      A     I 5.2;
      =     M 14.2;
      A     L 2.0;
      A     I 5.3;
      =     M 14.3;
      A     L 2.0;
      A     I 5.4;
      =     M 14.4;
      A     L 2.0;
      A     I 5.5;
      =     M 14.5;
      A     L 2.0;
      A     I 5.6;
      =     M 14.6;
      A     L 2.0;
      A     I 5.7;
      =     M 14.7;
      A     L 2.0;
      A     I 6.0;
      =     M 15.0;
      A     L 2.0;
      A     I 6.1;
      =     M 15.1;
      A     L 2.0;
      A     I 6.2;
      =     M 15.2;
      A     L 2.0;
      A     I 6.3;
      =     M 15.3;
      A     L 2.0;
      A     I 6.4;
      =     M 15.4;
      A     L 2.0;
      A     I 6.5;
      =     M 15.5;
      A     L 2.0;
      A     I 6.6;
      =     M 15.6;
      A     L 2.0;
      A(;
      O     I 6.7;
      O     M 1.1;
      );
      =     M 15.7;
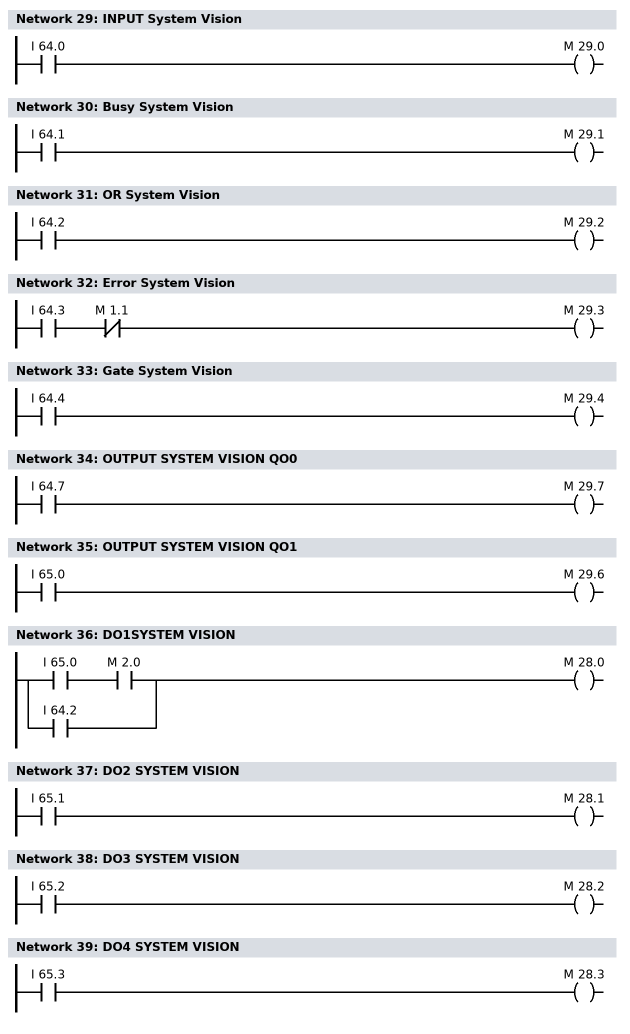
NETWORK
TITLE = INPUT System Vision 
      A     I 64.0;
      =     M 29.0;
NETWORK
TITLE = Busy System Vision
      A     I 64.1;
      =     M 29.1;
NETWORK
TITLE = OR System Vision
      A     I 64.2;
      =     M 29.2;
NETWORK
TITLE = Error System Vision
      A     I 64.3;
      AN    M 1.1;
      =     M 29.3;
NETWORK
TITLE = Gate System Vision
      A     I 64.4;
      =     M 29.4;
NETWORK
TITLE = OUTPUT SYSTEM VISION QO0
      A     I 64.7;
      =     M 29.7;
NETWORK
TITLE = OUTPUT SYSTEM VISION QO1
      A     I 65.0;
      =     M 29.6;
NETWORK
TITLE = DO1SYSTEM VISION
      A     I 65.0;
      A     M 2.0;
      O     I 64.2;
      =     M 28.0;
NETWORK
TITLE = DO2 SYSTEM VISION
      A     I 65.1;
      =     M 28.1;
NETWORK
TITLE = DO3 SYSTEM VISION
      A     I 65.2;
      =     M 28.2;
NETWORK
TITLE = DO4 SYSTEM VISION
      A     I 65.3;
      =     M 28.3;
END_FUNCTION

FUNCTION "FC12 - GENERAL" : VOID	// FC 12
TITLE = General management
VERSION : 0.1
BEGIN
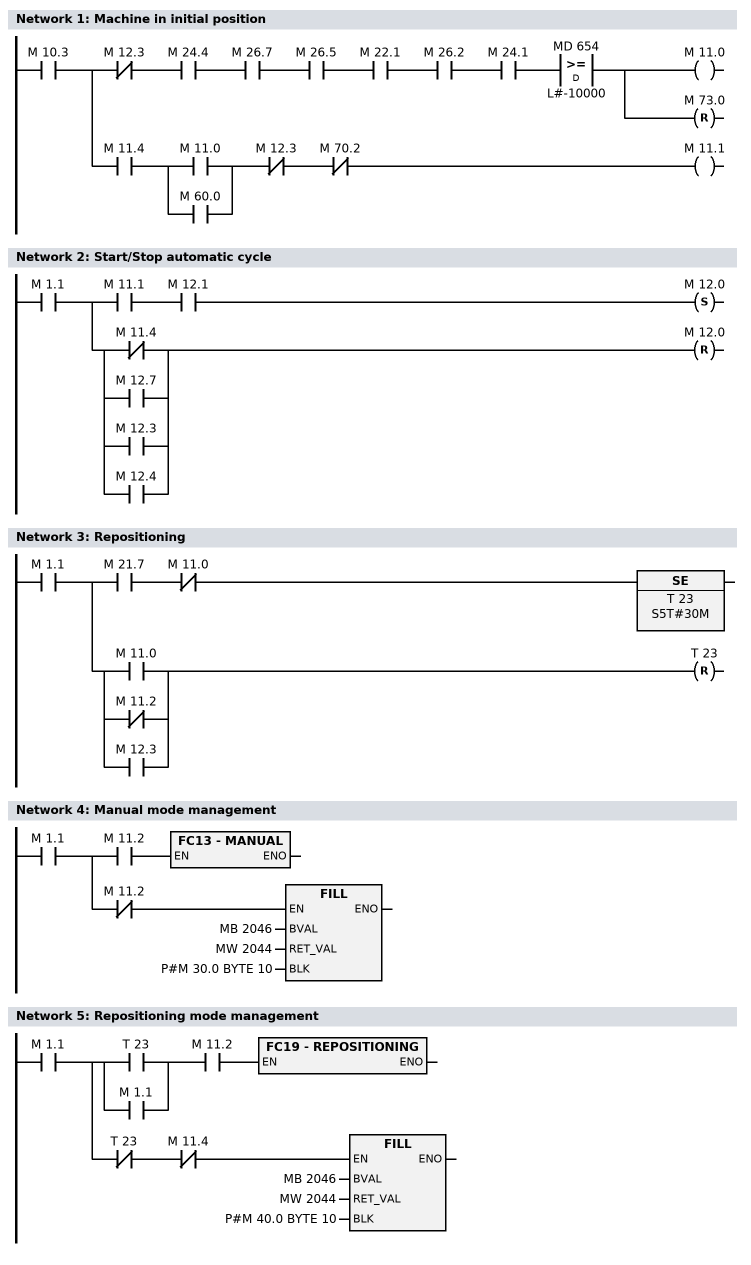
NETWORK
TITLE = Machine in initial position
      A     M 10.3;
      =     L 0.0;
      A     L 0.0;
      AN    M 12.3;
      A     M 24.4;
      A     M 26.7;
      A     M 26.5;
      A     M 22.1;
      A     M 26.2;
      A     M 24.1;
      A(;
      L     MD 654;
      L     L#-10000;
      >=D;
      );
      =     M 11.0;
      R     M 73.0;
      A     L 0.0;
      A     M 11.4;
      A(;
      O     M 11.0;
      O     M 60.0;
      );
      AN    M 12.3;
      AN    M 70.2;
      =     M 11.1;
NETWORK
TITLE = Start/Stop automatic cycle
      A     M 1.1;
      =     L 0.0;
      A     L 0.0;
      A     M 11.1;
      A     M 12.1;
      S     M 12.0;
      A     L 0.0;
      A(;
      ON    M 11.4;
      O     M 12.7;
      O     M 12.3;
      O     M 12.4;
      );
      R     M 12.0;
NETWORK
TITLE = Repositioning
      A     M 1.1;
      =     L 0.0;
      A     L 0.0;
      A     M 21.7;
      AN    M 11.0;
      L     S5T#30M;
      SE    T 23;
      A     L 0.0;
      A(;
      O     M 11.0;
      ON    M 11.2;
      O     M 12.3;
      );
      R     T 23;
NETWORK
TITLE = Manual mode management
      A     M 1.1;
      =     L 0.0;
      A     L 0.0;
      A     M 11.2;
      JNB   _001;
      CALL  "FC13 - MANUAL";
_001: NOP   0;
      A     L 0.0;
      AN    M 11.2;
      JNB   _002;
      CALL  "FILL" (
           BVAL                     := MB 2046,
           RET_VAL                  := MW 2044,
           BLK                      := P#M 30.0 BYTE 10);
_002: NOP   0;
NETWORK
TITLE = Repositioning mode management
      A     M 1.1;
      =     L 0.0;
      A     L 0.0;
      A(;
      O     T 23;
      O     M 1.1;
      );
      A     M 11.2;
      JNB   _003;
      CALL  "FC19 - REPOSITIONING";
_003: NOP   0;
      A     L 0.0;
      AN    T 23;
      AN    M 11.4;
      JNB   _004;
      CALL  "FILL" (
           BVAL                     := MB 2046,
           RET_VAL                  := MW 2044,
           BLK                      := P#M 40.0 BYTE 10);
_004: NOP   0;
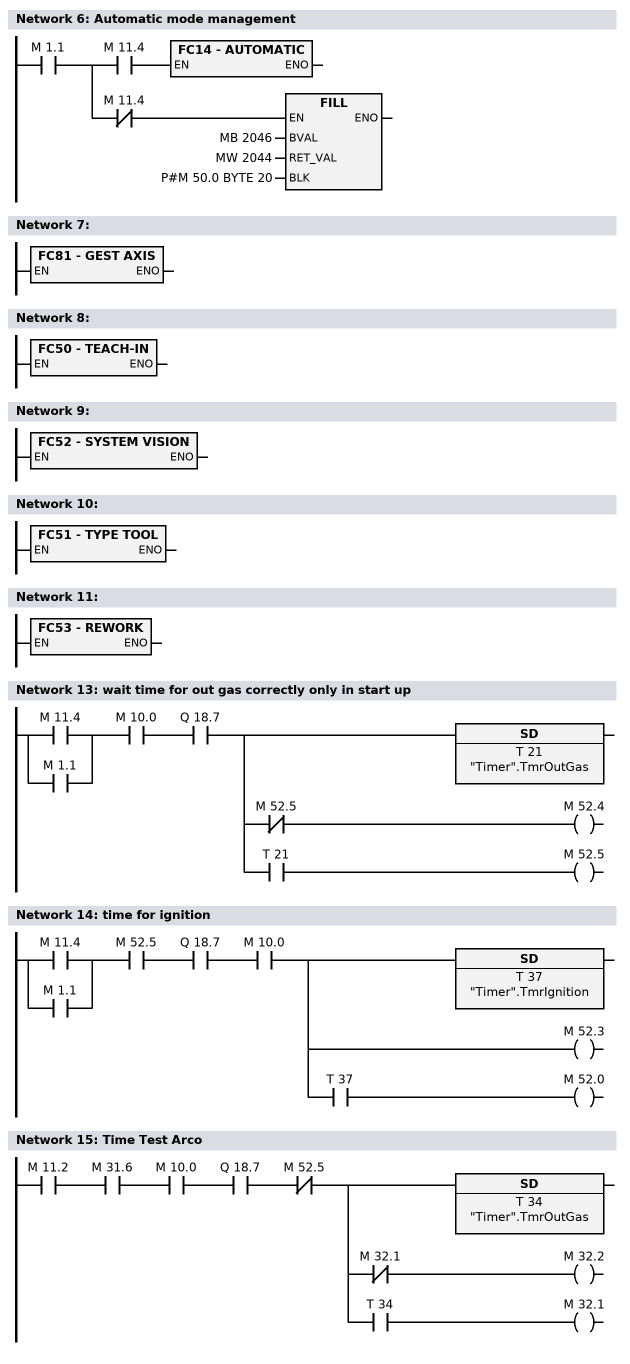
NETWORK
TITLE = Automatic mode management
//reset axis mouvement
      A     M 1.1;
      =     L 0.0;
      A     L 0.0;
      A     M 11.4;
      JNB   _005;
      CALL  "FC14 - AUTOMATIC";
_005: NOP   0;
      A     L 0.0;
      AN    M 11.4;
      JNB   _006;
      CALL  "FILL" (
           BVAL                     := MB 2046,
           RET_VAL                  := MW 2044,
           BLK                      := P#M 50.0 BYTE 20);
_006: NOP   0;
NETWORK
TITLE =
      CALL  "FC81 - GEST AXIS";
      NOP   0;
NETWORK
TITLE =
      CALL  "FC50 - TEACH-IN";
      NOP   0;
NETWORK
TITLE =
      CALL  "FC52 - SYSTEM VISION";
      NOP   0;
NETWORK
TITLE =
//Controllo il tipo di portapezzo e carico i relativi dati
      CALL  "FC51 - TYPE TOOL";
      NOP   0;
NETWORK
TITLE =
      CALL  "FC53 - REWORK";
      NOP   0;
NETWORK
TITLE =
NETWORK
TITLE = wait time for out gas correctly only in start up 
//AUT - Tempo di attesa per avere gas in circolo e la torcia in temp
      A(;
      O     M 11.4;
      O     M 1.1;
      );
      A     M 10.0;
      A     Q 18.7;
      =     L 0.0;
      A     L 0.0;
      BLD   102;
      L     "Timer".TmrOutGas;
      SD    T 21;
      A     L 0.0;
      AN    M 52.5;
      =     M 52.4;
      A     L 0.0;
      A     T 21;
      =     M 52.5;
NETWORK
TITLE = time for ignition
      A(;
      O     M 11.4;
      O     M 1.1;
      );
      A     M 52.5;
      A     Q 18.7;
      A     M 10.0;
      =     L 0.0;
      A     L 0.0;
      BLD   102;
      L     "Timer".TmrIgnition;
      SD    T 37;
      A     L 0.0;
      BLD   102;
      =     M 52.3;
      A     L 0.0;
      A     T 37;
      =     M 52.0;
NETWORK
TITLE = Time Test Arco
//Test Arco Gas in Manuale
      A     M 11.2;
      A     M 31.6;
      A     M 10.0;
      A     Q 18.7;
      AN    M 52.5;
      =     L 0.0;
      A     L 0.0;
      BLD   102;
      L     "Timer".TmrOutGas;
      SD    T 34;
      A     L 0.0;
      AN    M 32.1;
      =     M 32.2;
      A     L 0.0;
      A     T 34;
      =     M 32.1;
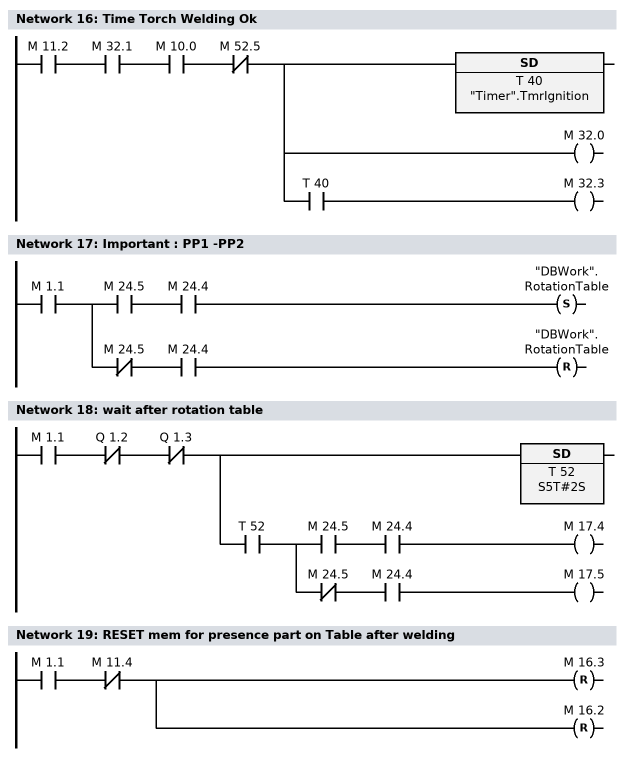
NETWORK
TITLE = Time Torch Welding Ok
//Accensione Torcia in Manuale: per arrivare in Temp
      A     M 11.2;
      A     M 32.1;
      A     M 10.0;
      AN    M 52.5;
      =     L 0.0;
      A     L 0.0;
      BLD   102;
      L     "Timer".TmrIgnition;
      SD    T 40;
      A     L 0.0;
      BLD   102;
      =     M 32.0;
      A     L 0.0;
      A     T 40;
      =     M 32.3;
NETWORK
TITLE = Important : PP1 -PP2 
      A     M 1.1;
      =     L 0.0;
      A     L 0.0;
      A     M 24.5;
      A     M 24.4;
      S     "DBWork".RotationTable;
      A     L 0.0;
      AN    M 24.5;
      A     M 24.4;
      R     "DBWork".RotationTable;
NETWORK
TITLE = wait after rotation table
      A     M 1.1;
      AN    Q 1.2;
      AN    Q 1.3;
      =     L 0.0;
      A     L 0.0;
      BLD   102;
      L     S5T#2S;
      SD    T 52;
      A     L 0.0;
      A     T 52;
      =     L 0.1;
      A     L 0.1;
      A     M 24.5;
      A     M 24.4;
      =     M 17.4;
      A     L 0.1;
      AN    M 24.5;
      A     M 24.4;
      =     M 17.5;
NETWORK
TITLE = RESET mem for presence part on Table after welding
      A     M 1.1;
      AN    M 11.4;
      R     M 16.3;
      R     M 16.2;
END_FUNCTION

FUNCTION "FC13 - MANUAL" : VOID	// FC 13
TITLE = Manual commands
VERSION : 0.1
BEGIN
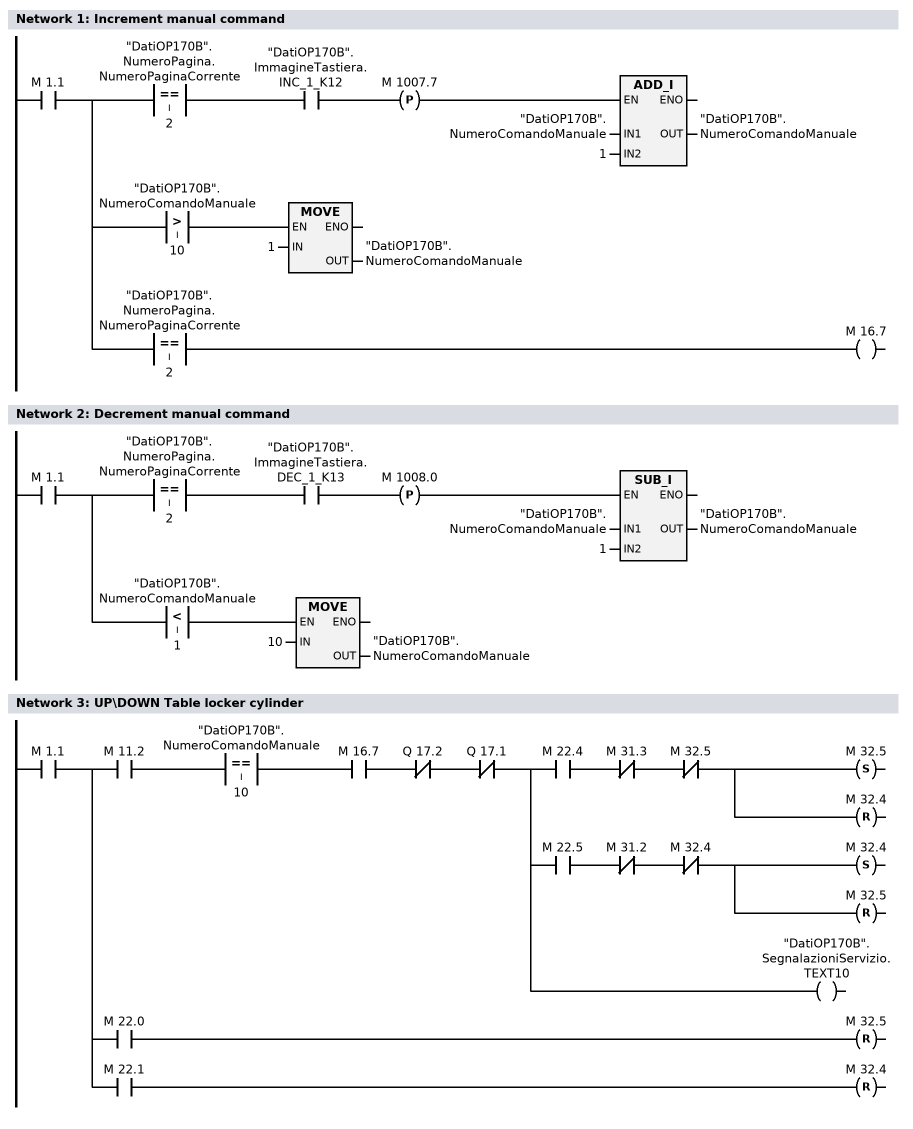
NETWORK
TITLE = Increment manual command
      A     M 1.1;
      =     L 1.0;
      A     L 1.0;
      A(;
      L     "DatiOP170B".NumeroPagina.NumeroPaginaCorrente;
      L     2;
      ==I;
      );
      A     "DatiOP170B".ImmagineTastiera.INC_1_K12;
      FP    M 1007.7;
      JNB   _001;
      L     "DatiOP170B".NumeroComandoManuale;
      L     1;
      +I;
      T     "DatiOP170B".NumeroComandoManuale;
_001: NOP   0;
      A     L 1.0;
      A(;
      L     "DatiOP170B".NumeroComandoManuale;
      L     10;
      >I;
      );
      JNB   _002;
      L     1;
      T     "DatiOP170B".NumeroComandoManuale;
_002: NOP   0;
      A     L 1.0;
      A(;
      L     "DatiOP170B".NumeroPagina.NumeroPaginaCorrente;
      L     2;
      ==I;
      );
      =     M 16.7;
NETWORK
TITLE = Decrement manual command
      A     M 1.1;
      =     L 1.0;
      A     L 1.0;
      A(;
      L     "DatiOP170B".NumeroPagina.NumeroPaginaCorrente;
      L     2;
      ==I;
      );
      A     "DatiOP170B".ImmagineTastiera.DEC_1_K13;
      FP    M 1008.0;
      JNB   _003;
      L     "DatiOP170B".NumeroComandoManuale;
      L     1;
      -I;
      T     "DatiOP170B".NumeroComandoManuale;
_003: NOP   0;
      A     L 1.0;
      A(;
      L     "DatiOP170B".NumeroComandoManuale;
      L     1;
      <I;
      );
      JNB   _004;
      L     10;
      T     "DatiOP170B".NumeroComandoManuale;
_004: NOP   0;
NETWORK
TITLE = UP\DOWN Table locker cylinder
      A     M 1.1;
      =     L 1.0;
      A     L 1.0;
      A     M 11.2;
      A(;
      L     "DatiOP170B".NumeroComandoManuale;
      L     10;
      ==I;
      );
      A     M 16.7;
      AN    Q 17.2;
      AN    Q 17.1;
      =     L 1.1;
      A     L 1.1;
      A     M 22.4;
      AN    M 31.3;
      AN    M 32.5;
      S     M 32.5;
      R     M 32.4;
      A     L 1.1;
      A     M 22.5;
      AN    M 31.2;
      AN    M 32.4;
      S     M 32.4;
      R     M 32.5;
      A     L 1.1;
      BLD   102;
      =     "DatiOP170B".SegnalazioniServizio.TEXT10;
      A     L 1.0;
      A     M 22.0;
      R     M 32.5;
      A     L 1.0;
      A     M 22.1;
      R     M 32.4;
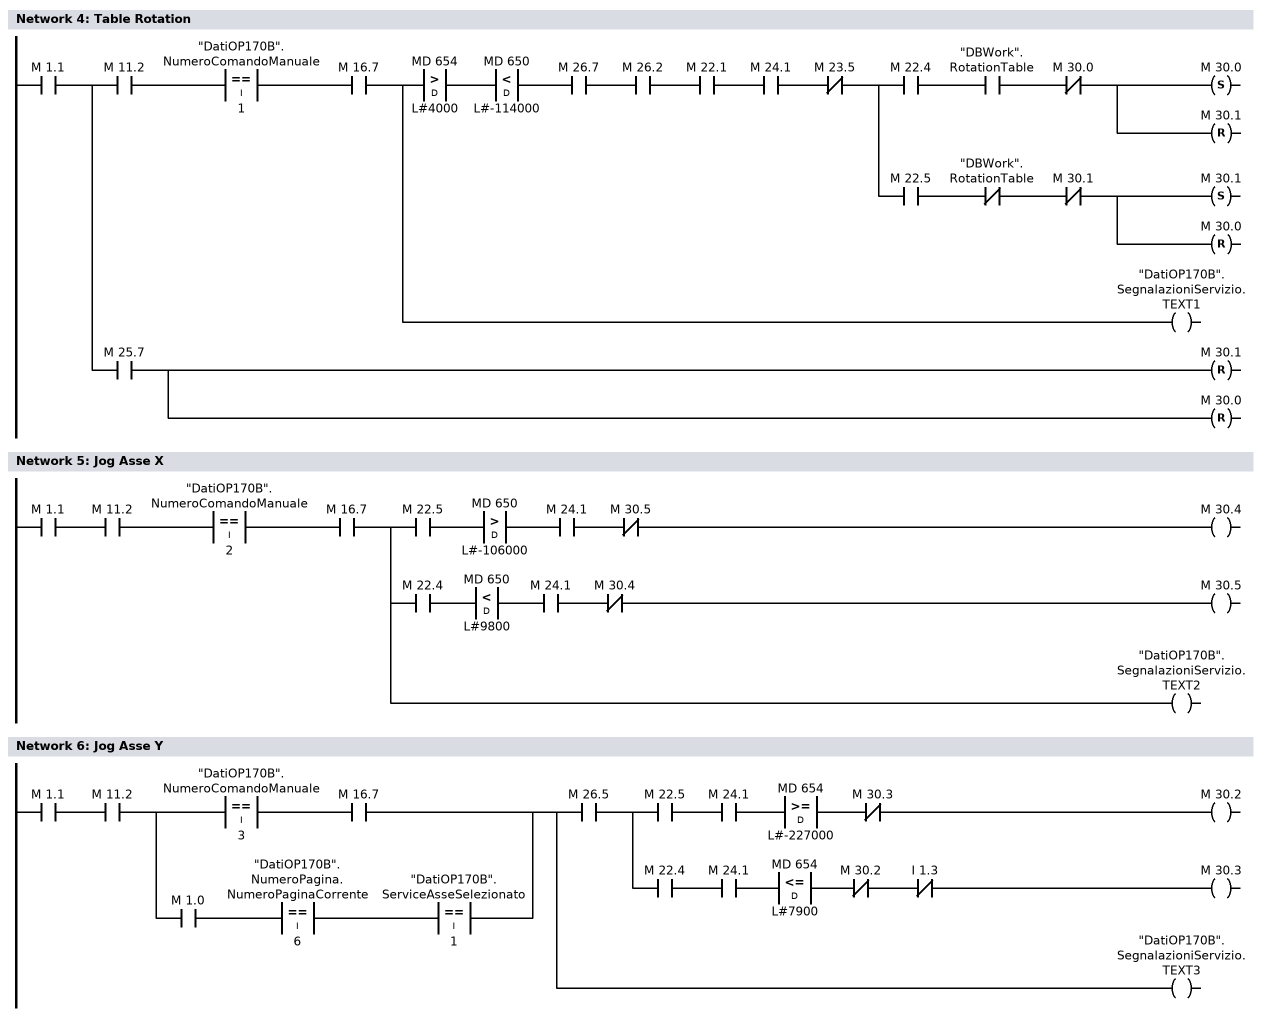
NETWORK
TITLE = Table Rotation
      A     M 1.1;
      =     L 1.0;
      A     L 1.0;
      A     M 11.2;
      A(;
      L     "DatiOP170B".NumeroComandoManuale;
      L     1;
      ==I;
      );
      A     M 16.7;
      =     L 1.1;
      A     L 1.1;
      A(;
      L     MD 654;
      L     L#4000;
      >D;
      );
      A(;
      L     MD 650;
      L     L#-114000;
      <D;
      );
      A     M 26.7;
      A     M 26.2;
      A     M 22.1;
      A     M 24.1;
      AN    M 23.5;
      =     L 1.2;
      A     L 1.2;
      A     M 22.4;
      A     "DBWork".RotationTable;
      AN    M 30.0;
      S     M 30.0;
      R     M 30.1;
      A     L 1.2;
      A     M 22.5;
      AN    "DBWork".RotationTable;
      AN    M 30.1;
      S     M 30.1;
      R     M 30.0;
      A     L 1.1;
      BLD   102;
      =     "DatiOP170B".SegnalazioniServizio.TEXT1;
      A     L 1.0;
      A     M 25.7;
      R     M 30.1;
      R     M 30.0;
NETWORK
TITLE = Jog Asse X
      A     M 1.1;
      A     M 11.2;
      A(;
      A(;
      L     "DatiOP170B".NumeroComandoManuale;
      L     2;
      ==I;
      );
      A     M 16.7;
      );
      =     L 0.0;
      A     L 0.0;
      A     M 22.5;
      A(;
      L     MD 650;
      L     L#-106000;
      >D;
      );
      A     M 24.1;
      AN    M 30.5;
      =     M 30.4;
      A     L 0.0;
      A     M 22.4;
      A(;
      L     MD 650;
      L     L#9800;
      <D;
      );
      A     M 24.1;
      AN    M 30.4;
      =     M 30.5;
      A     L 0.0;
      BLD   102;
      =     "DatiOP170B".SegnalazioniServizio.TEXT2;
NETWORK
TITLE = Jog Asse Y
      A     M 1.1;
      A     M 11.2;
      A(;
      A(;
      L     "DatiOP170B".NumeroComandoManuale;
      L     3;
      ==I;
      );
      A     M 16.7;
      O;
      A     M 1.0;
      A(;
      L     "DatiOP170B".NumeroPagina.NumeroPaginaCorrente;
      L     6;
      ==I;
      );
      A(;
      L     "DatiOP170B".ServiceAsseSelezionato;
      L     1;
      ==I;
      );
      );
      =     L 0.0;
      A     L 0.0;
      A     M 26.5;
      =     L 0.1;
      A     L 0.1;
      A     M 22.5;
      A     M 24.1;
      A(;
      L     MD 654;
      L     L#-227000;
      >=D;
      );
      AN    M 30.3;
      =     M 30.2;
      A     L 0.1;
      A     M 22.4;
      A     M 24.1;
      A(;
      L     MD 654;
      L     L#7900;
      <=D;
      );
      AN    M 30.2;
      AN    I 1.3;
      =     M 30.3;
      A     L 0.0;
      BLD   102;
      =     "DatiOP170B".SegnalazioniServizio.TEXT3;
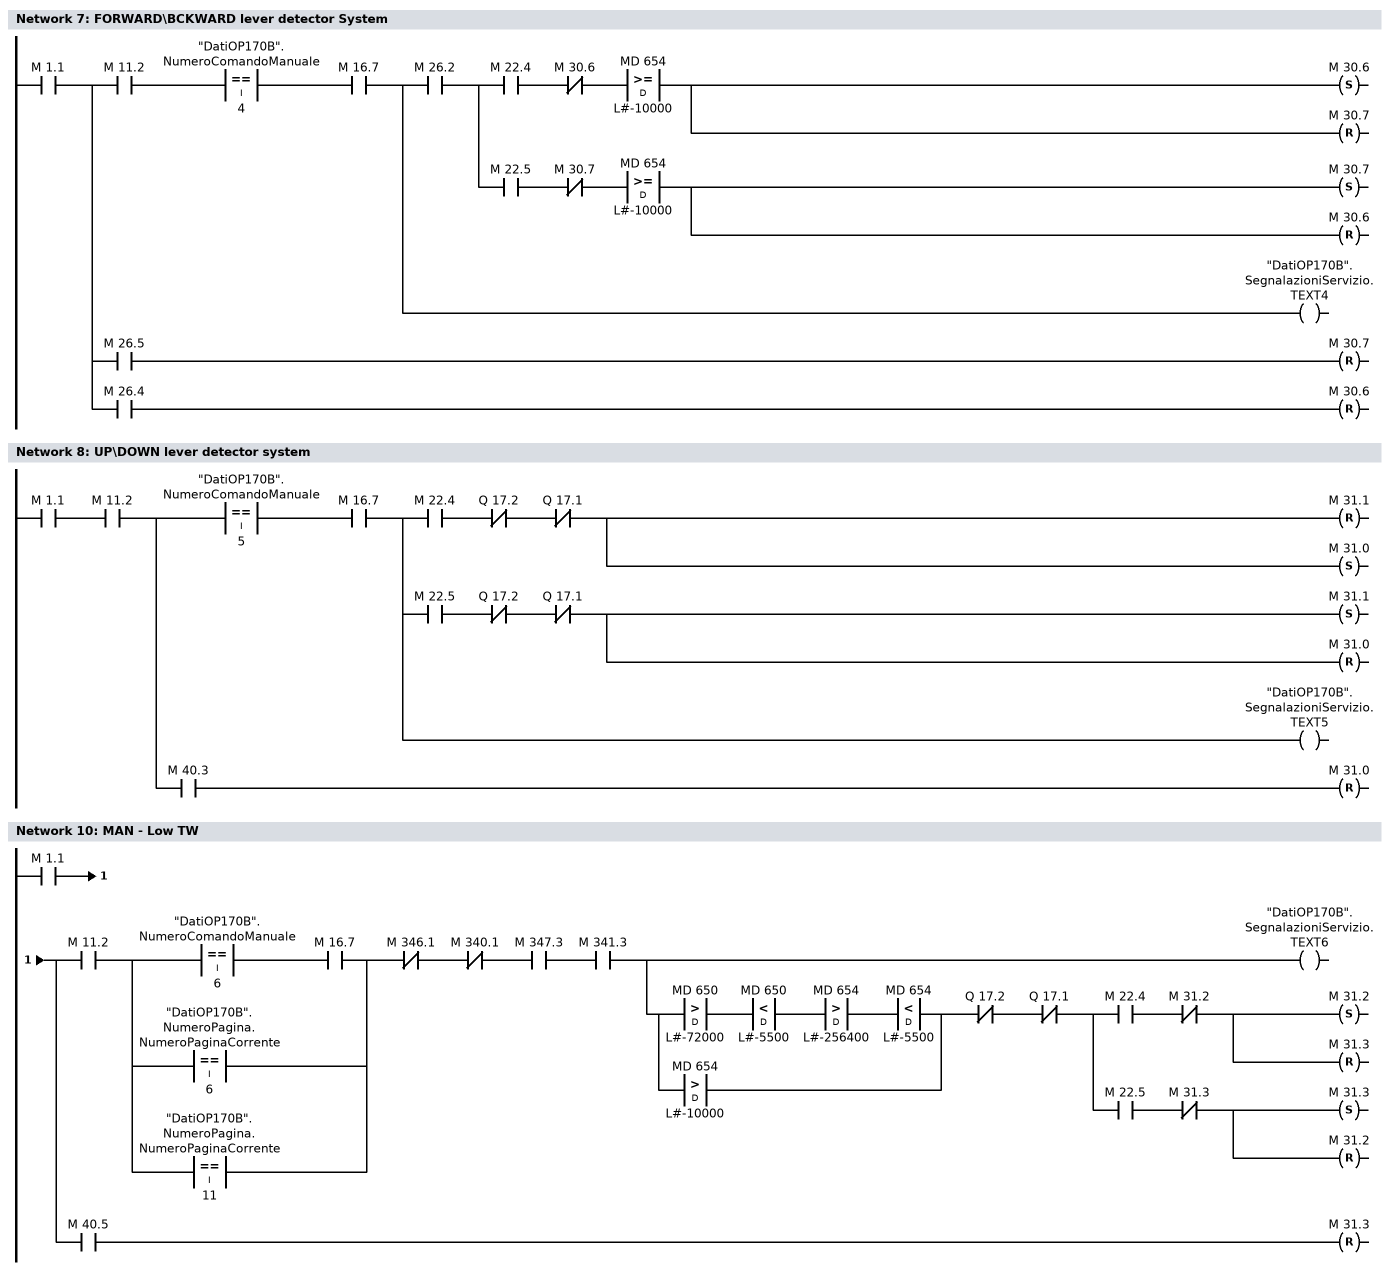
NETWORK
TITLE = FORWARD\BCKWARD lever detector System
//controllo fuori ingombro asse Y
      A     M 1.1;
      =     L 1.0;
      A     L 1.0;
      A     M 11.2;
      A(;
      L     "DatiOP170B".NumeroComandoManuale;
      L     4;
      ==I;
      );
      A     M 16.7;
      =     L 1.1;
      A     L 1.1;
      A     M 26.2;
      =     L 1.2;
      A     L 1.2;
      A     M 22.4;
      AN    M 30.6;
      A(;
      L     MD 654;
      L     L#-10000;
      >=D;
      );
      S     M 30.6;
      R     M 30.7;
      A     L 1.2;
      A     M 22.5;
      AN    M 30.7;
      A(;
      L     MD 654;
      L     L#-10000;
      >=D;
      );
      S     M 30.7;
      R     M 30.6;
      A     L 1.1;
      BLD   102;
      =     "DatiOP170B".SegnalazioniServizio.TEXT4;
      A     L 1.0;
      A     M 26.5;
      R     M 30.7;
      A     L 1.0;
      A     M 26.4;
      R     M 30.6;
NETWORK
TITLE = UP\DOWN lever detector system
      A     M 1.1;
      A     M 11.2;
      =     L 1.0;
      A     L 1.0;
      A(;
      L     "DatiOP170B".NumeroComandoManuale;
      L     5;
      ==I;
      );
      A     M 16.7;
      =     L 1.1;
      A     L 1.1;
      A     M 22.4;
      AN    Q 17.2;
      AN    Q 17.1;
      R     M 31.1;
      S     M 31.0;
      A     L 1.1;
      A     M 22.5;
      AN    Q 17.2;
      AN    Q 17.1;
      S     M 31.1;
      R     M 31.0;
      A     L 1.1;
      BLD   102;
      =     "DatiOP170B".SegnalazioniServizio.TEXT5;
      A     L 1.0;
      A     M 40.3;
      R     M 31.0;
NETWORK
TITLE = UP\DOWN Torch Welding Machine
//      U     "On"
//      =     L      0.0
//      U     L      0.0
//      U     "M11.2"
//      U(    
//      U(    
//      L     "DatiOP170B".NumeroComandoManuale
//      L     6
//      ==I   
//      )     
//      U     "M16.7"
//      O     
//      U(    
//      O(    
//      L     "DatiOP170B".NumeroPagina.NumeroPaginaCorrente
//      L     6
//      ==I   
//      )     
//      O(    
//      L     "DatiOP170B".NumeroPagina.NumeroPaginaCorrente
//      L     11
//      ==I   
//      )     
//      )     
//      UN    "M346.1"
//      UN    "M340.1"
//      U     "M347.3"
//      U     "M341.3"
//      )     
//      =     L      0.1
//      U     L      0.1
//      U(    
//      U(    
//      L     "MD650"
//      L     L#-72000
//      >D    
//      )     
//      U(    
//      L     "MD650"
//      L     L#-5500
//      <D    
//      )     
//      U(    
//      L     "MD654"
//      L     L#-256400
//      >D    
//      )     
//      U(    
//      L     "MD654"
//      L     L#-5500
//      <D    
//      )     
//      O(    
//      L     "MD654"
//      L     -10000
//      >D    
//      )     
//      )     
//      UN    "REVERSE_TABLE_ROTATION"
//      UN    "FWD_TABLE_ROTATION"
//      =     L      0.2
//      U     L      0.2
//      U     "M22.4"
//      UN    "M31.2"
//      S     "M31.2"
//      R     "M31.3"
//      U     L      0.2
//      U     "M22.5"
//      UN    "M31.3"
//      S     "M31.3"
//      R     "M31.2"
//      U     L      0.1
//      BLD   102
//      =     "DatiOP170B".SegnalazioniServizio.TEXT6
//      U     L      0.0
//      U     "M40.5"
//      R     "M31.3"
//  A     L      0.0
// A     "M24.1"
// R     "M31.2"
NETWORK
TITLE = MAN - Low TW
      A     M 1.1;
      =     L 1.0;
      A     L 1.0;
      A     M 11.2;
      A(;
      A(;
      L     "DatiOP170B".NumeroComandoManuale;
      L     6;
      ==I;
      );
      A     M 16.7;
      O(;
      L     "DatiOP170B".NumeroPagina.NumeroPaginaCorrente;
      L     6;
      ==I;
      );
      O(;
      L     "DatiOP170B".NumeroPagina.NumeroPaginaCorrente;
      L     11;
      ==I;
      );
      );
      AN    M 346.1;
      AN    M 340.1;
      A     M 347.3;
      A     M 341.3;
      =     L 1.1;
      A     L 1.1;
      BLD   102;
      =     "DatiOP170B".SegnalazioniServizio.TEXT6;
      A     L 1.1;
      A(;
      A(;
      L     MD 650;
      L     L#-72000;
      >D;
      );
      A(;
      L     MD 650;
      L     L#-5500;
      <D;
      );
      A(;
      L     MD 654;
      L     L#-256400;
      >D;
      );
      A(;
      L     MD 654;
      L     L#-5500;
      <D;
      );
      O(;
      L     MD 654;
      L     L#-10000;
      >D;
      );
      );
      AN    Q 17.2;
      AN    Q 17.1;
      =     L 1.2;
      A     L 1.2;
      A     M 22.4;
      AN    M 31.2;
      S     M 31.2;
      R     M 31.3;
      A     L 1.2;
      A     M 22.5;
      AN    M 31.3;
      S     M 31.3;
      R     M 31.2;
      A     L 1.0;
      A     M 40.5;
      R     M 31.3;
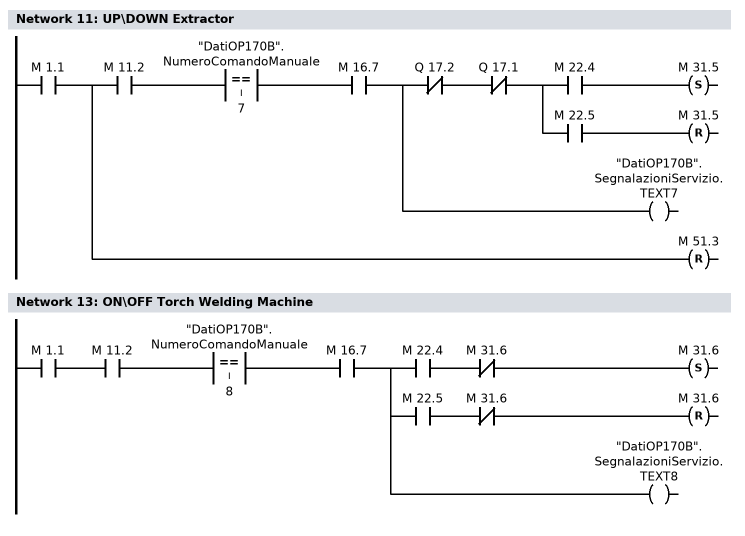
NETWORK
TITLE = UP\DOWN Extractor
      A     M 1.1;
      =     L 1.0;
      A     L 1.0;
      A     M 11.2;
      A(;
      L     "DatiOP170B".NumeroComandoManuale;
      L     7;
      ==I;
      );
      A     M 16.7;
      =     L 1.1;
      A     L 1.1;
      AN    Q 17.2;
      AN    Q 17.1;
      =     L 1.2;
      A     L 1.2;
      A     M 22.4;
      S     M 31.5;
      A     L 1.2;
      A     M 22.5;
      R     M 31.5;
      A     L 1.1;
      BLD   102;
      =     "DatiOP170B".SegnalazioniServizio.TEXT7;
      A     L 1.0;
      BLD   102;
      R     M 51.3;
NETWORK
TITLE =
NETWORK
TITLE = ON\OFF Torch Welding Machine
      A     M 1.1;
      A     M 11.2;
      A(;
      L     "DatiOP170B".NumeroComandoManuale;
      L     8;
      ==I;
      );
      A     M 16.7;
      =     L 1.0;
      A     L 1.0;
      A     M 22.4;
      AN    M 31.6;
      S     M 31.6;
      A     L 1.0;
      A     M 22.5;
      AN    M 31.6;
      R     M 31.6;
      A     L 1.0;
      BLD   102;
      =     "DatiOP170B".SegnalazioniServizio.TEXT8;
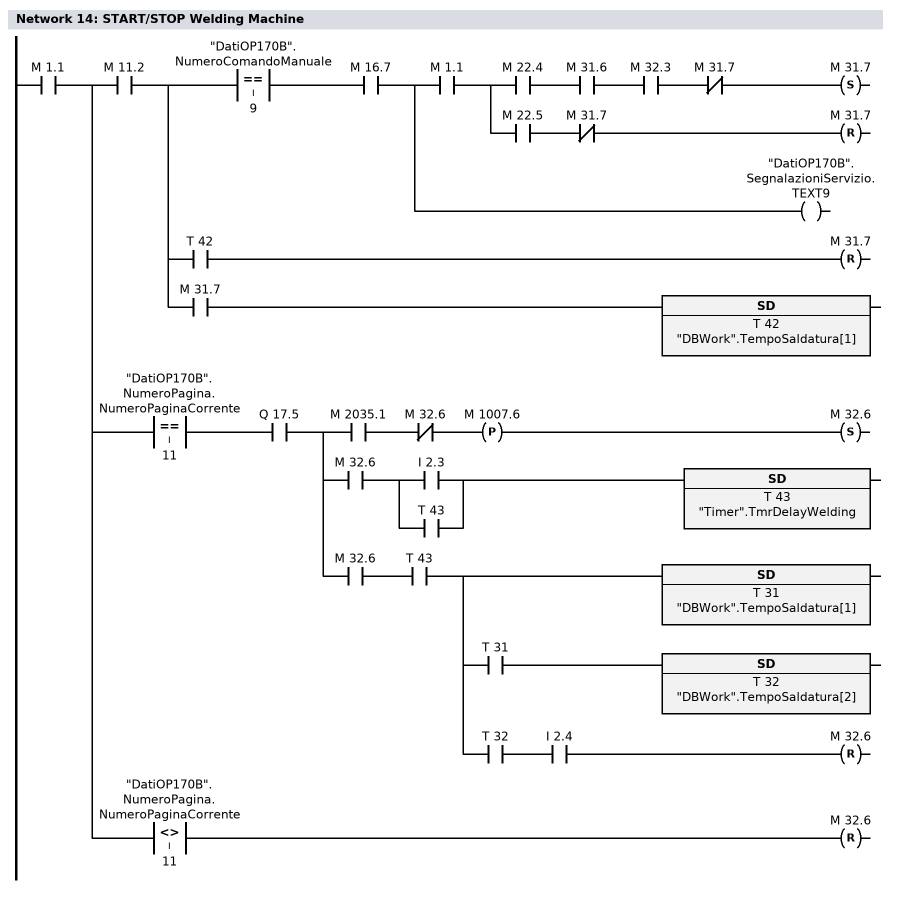
NETWORK
TITLE = START/STOP Welding Machine
      A     M 1.1;
      =     L 1.0;
      A     L 1.0;
      A     M 11.2;
      =     L 1.1;
      A     L 1.1;
      A(;
      L     "DatiOP170B".NumeroComandoManuale;
      L     9;
      ==I;
      );
      A     M 16.7;
      =     L 1.2;
      A     L 1.2;
      A     M 1.1;
      =     L 1.3;
      A     L 1.3;
      A     M 22.4;
      A     M 31.6;
      A     M 32.3;
      AN    M 31.7;
      S     M 31.7;
      A     L 1.3;
      A     M 22.5;
      AN    M 31.7;
      R     M 31.7;
      A     L 1.2;
      BLD   102;
      =     "DatiOP170B".SegnalazioniServizio.TEXT9;
      A     L 1.1;
      A     T 42;
      R     M 31.7;
      A     L 1.1;
      A     M 31.7;
      L     "DBWork".TempoSaldatura[1];
      SD    T 42;
      A     L 1.0;
      A(;
      L     "DatiOP170B".NumeroPagina.NumeroPaginaCorrente;
      L     11;
      ==I;
      );
      A     Q 17.5;
      =     L 1.1;
      A     L 1.1;
      A     M 2035.1;
      AN    M 32.6;
      FP    M 1007.6;
      S     M 32.6;
      A     L 1.1;
      A     M 32.6;
      A(;
      O     I 2.3;
      O     T 43;
      );
      L     "Timer".TmrDelayWelding;
      SD    T 43;
      A     L 1.1;
      A     M 32.6;
      A     T 43;
      =     L 1.2;
      A     L 1.2;
      BLD   102;
      L     "DBWork".TempoSaldatura[1];
      SD    T 31;
      A     L 1.2;
      A     T 31;
      L     "DBWork".TempoSaldatura[2];
      SD    T 32;
      A     L 1.2;
      A     T 32;
      A     I 2.4;
      R     M 32.6;
      A     L 1.0;
      A(;
      L     "DatiOP170B".NumeroPagina.NumeroPaginaCorrente;
      L     11;
      <>I;
      );
      R     M 32.6;
END_FUNCTION

FUNCTION "FC14 - AUTOMATIC" : VOID	// FC 14
TITLE = Automatic cycle management
VERSION : 0.1
VAR_TEMP
  MinX : DINT ;
  MinY : DINT ;
  MaxX : DINT ;
  MaxY : DINT ;
END_VAR
BEGIN
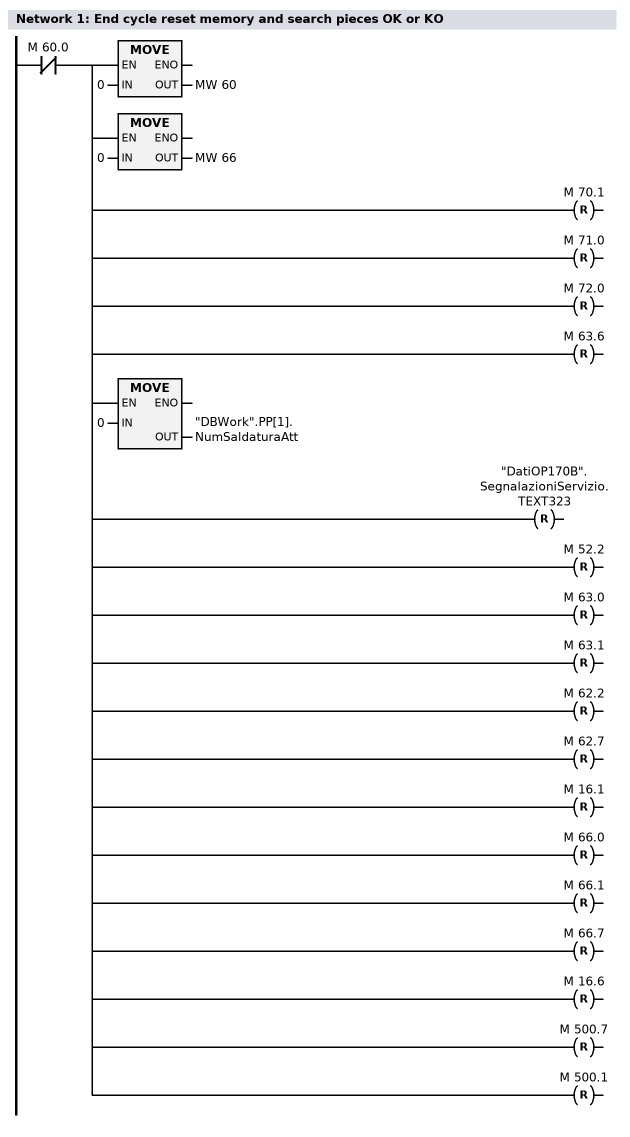
NETWORK
TITLE = End cycle reset memory and search pieces OK or KO
      AN    M 60.0;
      =     L 16.0;
      A     L 16.0;
      JNB   _001;
      L     0;
      T     MW 60;
_001: NOP   0;
      A     L 16.0;
      JNB   _002;
      L     0;
      T     MW 66;
_002: NOP   0;
      A     L 16.0;
      BLD   102;
      R     M 70.1;
      A     L 16.0;
      BLD   102;
      R     M 71.0;
      A     L 16.0;
      BLD   102;
      R     M 72.0;
      A     L 16.0;
      BLD   102;
      R     M 63.6;
      A     L 16.0;
      JNB   _003;
      L     0;
      T     "DBWork".PP[1].NumSaldaturaAtt;
_003: NOP   0;
      A     L 16.0;
      BLD   102;
      R     "DatiOP170B".SegnalazioniServizio.TEXT323;
      A     L 16.0;
      BLD   102;
      R     M 52.2;
      A     L 16.0;
      BLD   102;
      R     M 63.0;
      A     L 16.0;
      BLD   102;
      R     M 63.1;
      A     L 16.0;
      BLD   102;
      R     M 62.2;
      A     L 16.0;
      BLD   102;
      R     M 62.7;
      A     L 16.0;
      BLD   102;
      R     M 16.1;
      A     L 16.0;
      BLD   102;
      R     M 66.0;
      A     L 16.0;
      BLD   102;
      R     M 66.1;
      A     L 16.0;
      BLD   102;
      R     M 66.7;
      A     L 16.0;
      BLD   102;
      R     M 16.6;
      A     L 16.0;
      BLD   102;
      R     M 500.7;
      A     L 16.0;
      BLD   102;
      R     M 500.1;
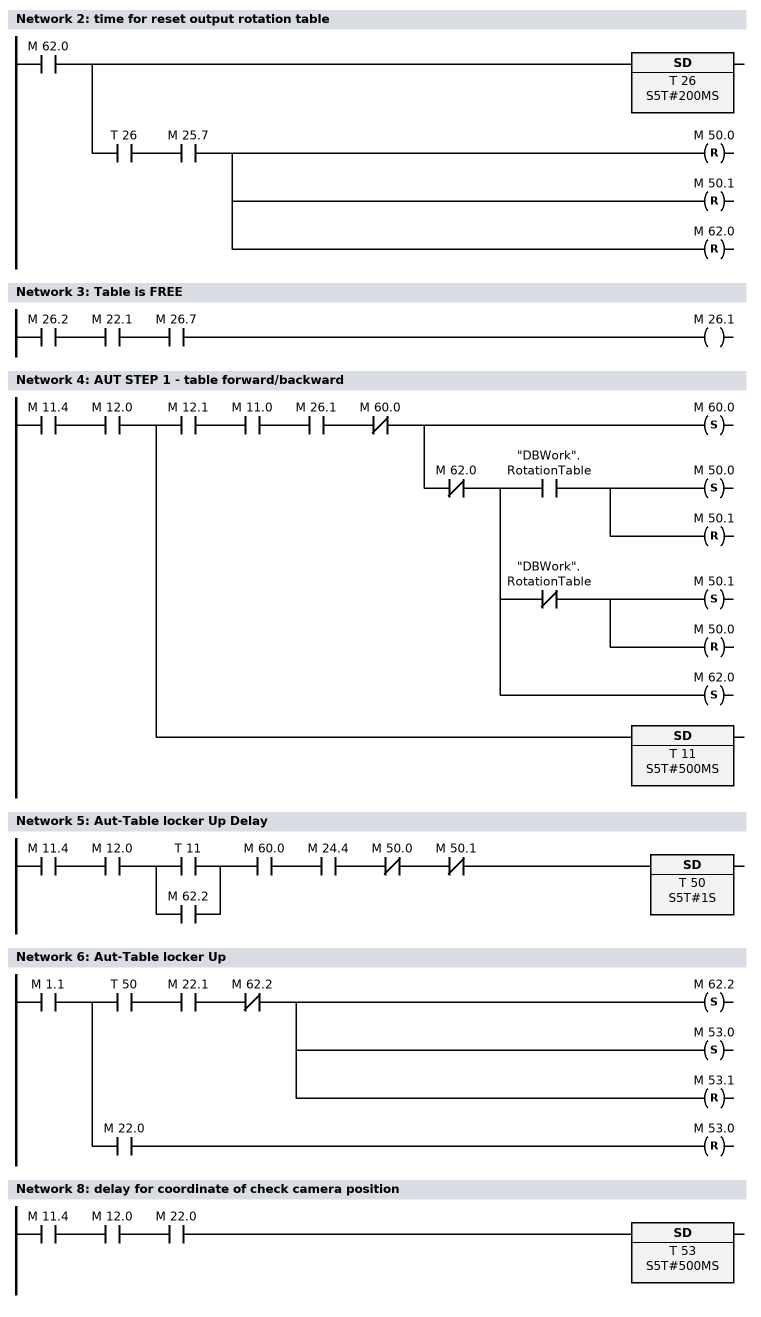
NETWORK
TITLE = time for reset output rotation table
//Reset Output Rotation Table 
      A     M 62.0;
      =     L 16.0;
      A     L 16.0;
      BLD   102;
      L     S5T#200MS;
      SD    T 26;
      A     L 16.0;
      A     T 26;
      A     M 25.7;
      R     M 50.0;
      R     M 50.1;
      R     M 62.0;
NETWORK
TITLE = Table is FREE
      A     M 26.2;
      A     M 22.1;
      A     M 26.7;
      =     M 26.1;
NETWORK
TITLE = AUT STEP 1 - table forward/backward
      A     M 11.4;
      A     M 12.0;
      =     L 16.0;
      A     L 16.0;
      A     M 12.1;
      A     M 11.0;
      A     M 26.1;
      AN    M 60.0;
      =     L 16.1;
      A     L 16.1;
      BLD   102;
      S     M 60.0;
      A     L 16.1;
      AN    M 62.0;
      =     L 16.2;
      A     L 16.2;
      A     "DBWork".RotationTable;
      S     M 50.0;
      R     M 50.1;
      A     L 16.2;
      AN    "DBWork".RotationTable;
      S     M 50.1;
      R     M 50.0;
      A     L 16.2;
      BLD   102;
      S     M 62.0;
      A     L 16.0;
      BLD   102;
      L     S5T#500MS;
      SD    T 11;
NETWORK
TITLE = Aut-Table locker Up Delay
      A     M 11.4;
      A     M 12.0;
      A(;
      O     T 11;
      O     M 62.2;
      );
      A     M 60.0;
      A     M 24.4;
      AN    M 50.0;
      AN    M 50.1;
      L     S5T#1S;
      SD    T 50;
NETWORK
TITLE = Aut-Table locker Up
      A     M 1.1;
      =     L 16.0;
      A     L 16.0;
      A     T 50;
      A     M 22.1;
      AN    M 62.2;
      S     M 62.2;
      S     M 53.0;
      R     M 53.1;
      A     L 16.0;
      A     M 22.0;
      R     M 53.0;
NETWORK
TITLE = Check With OMRON if Component is OK
NETWORK
TITLE = delay for coordinate of check camera position
      A     M 11.4;
      A     M 12.0;
      A     M 22.0;
      L     S5T#500MS;
      SD    T 53;
NETWORK
TITLE =
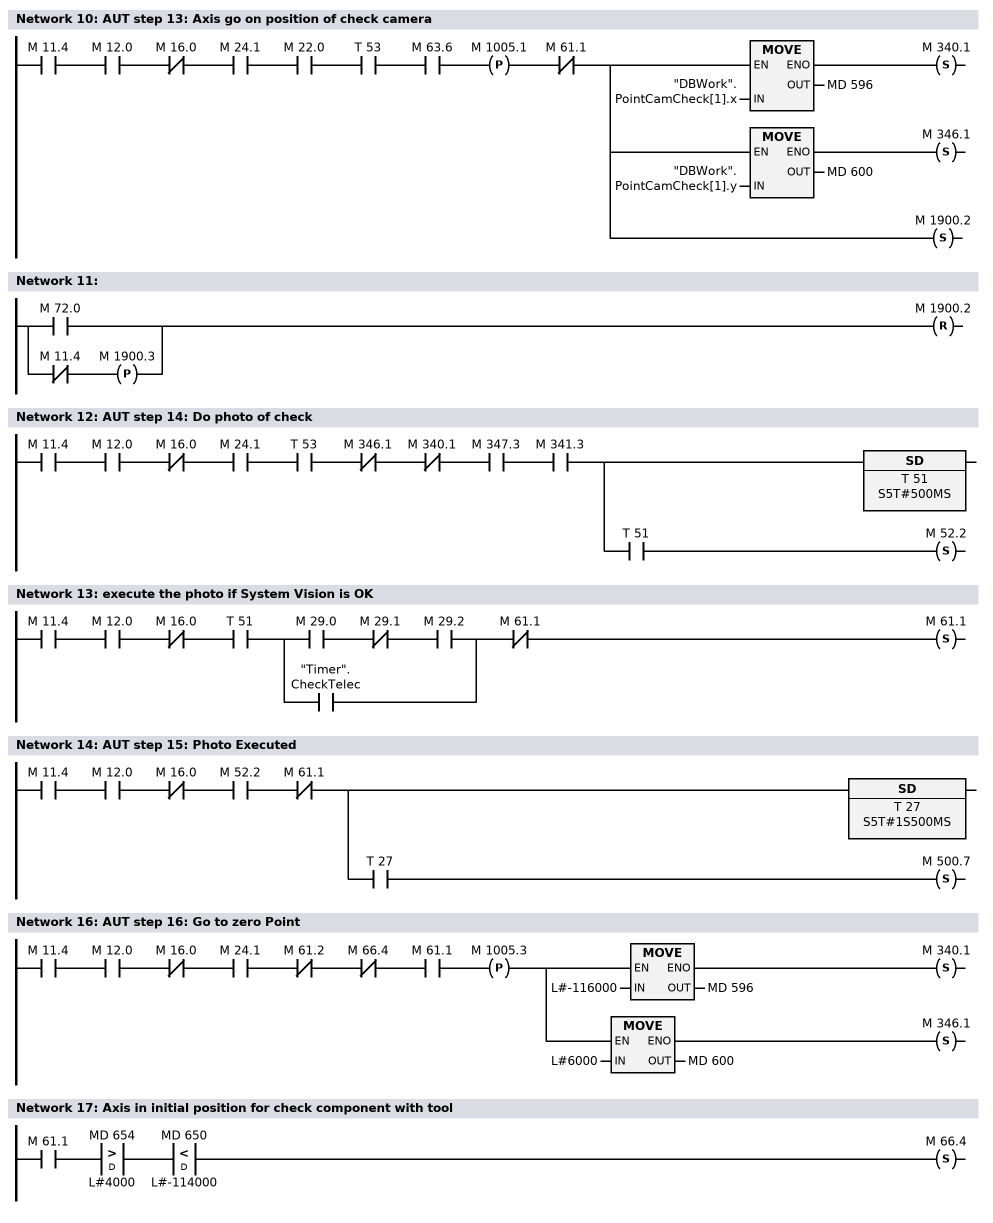
NETWORK
TITLE = AUT step 13: Axis go on position of check camera
      A     M 11.4;
      A     M 12.0;
      AN    M 16.0;
      A     M 24.1;
      A     M 22.0;
      A     T 53;
      A     M 63.6;
      FP    M 1005.1;
      AN    M 61.1;
      =     L 16.0;
      A     L 16.0;
      JNB   _004;
      L     "DBWork".PointCamCheck[1].x;
      T     MD 596;
      SET;
      SAVE;
      CLR;
_004: A     BR;
      S     M 340.1;
      A     L 16.0;
      JNB   _005;
      L     "DBWork".PointCamCheck[1].y;
      T     MD 600;
      SET;
      SAVE;
      CLR;
_005: A     BR;
      S     M 346.1;
      A     L 16.0;
      BLD   102;
      S     M 1900.2;
NETWORK
TITLE =
      O     M 72.0;
      O(;
      AN    M 11.4;
      FP    M 1900.3;
      );
      R     M 1900.2;
NETWORK
TITLE = AUT step 14: Do photo of check 
      A     M 11.4;
      A     M 12.0;
      AN    M 16.0;
      A     M 24.1;
      A     T 53;
      AN    M 346.1;
      AN    M 340.1;
      A     M 347.3;
      A     M 341.3;
      =     L 16.0;
      A     L 16.0;
      BLD   102;
      L     S5T#500MS;
      SD    T 51;
      A     L 16.0;
      A     T 51;
      S     M 52.2;
NETWORK
TITLE = execute the photo if System Vision is OK
      A     M 11.4;
      A     M 12.0;
      AN    M 16.0;
      A     T 51;
      A(;
      A     M 29.0;
      AN    M 29.1;
      A     M 29.2;
      O     "Timer".CheckTelec;
      );
      AN    M 61.1;
      S     M 61.1;
NETWORK
TITLE = AUT step 15: Photo Executed
      A     M 11.4;
      A     M 12.0;
      AN    M 16.0;
      A     M 52.2;
      AN    M 61.1;
      =     L 16.0;
      A     L 16.0;
      BLD   102;
      L     S5T#1S500MS;
      SD    T 27;
      A     L 16.0;
      A     T 27;
      S     M 500.7;
NETWORK
TITLE =
NETWORK
TITLE = AUT step 16: Go to zero Point
      A     M 11.4;
      A     M 12.0;
      AN    M 16.0;
      A     M 24.1;
      AN    M 61.2;
      AN    M 66.4;
      A     M 61.1;
      FP    M 1005.3;
      =     L 16.0;
      A     L 16.0;
      JNB   _006;
      L     L#-116000;
      T     MD 596;
      SET;
      SAVE;
      CLR;
_006: A     BR;
      S     M 340.1;
      A     L 16.0;
      JNB   _007;
      L     L#6000;
      T     MD 600;
      SET;
      SAVE;
      CLR;
_007: A     BR;
      S     M 346.1;
NETWORK
TITLE = Axis in initial position for check component with tool
      A     M 61.1;
      A(;
      L     MD 654;
      L     L#4000;
      >D;
      );
      A(;
      L     MD 650;
      L     L#-114000;
      <D;
      );
      S     M 66.4;
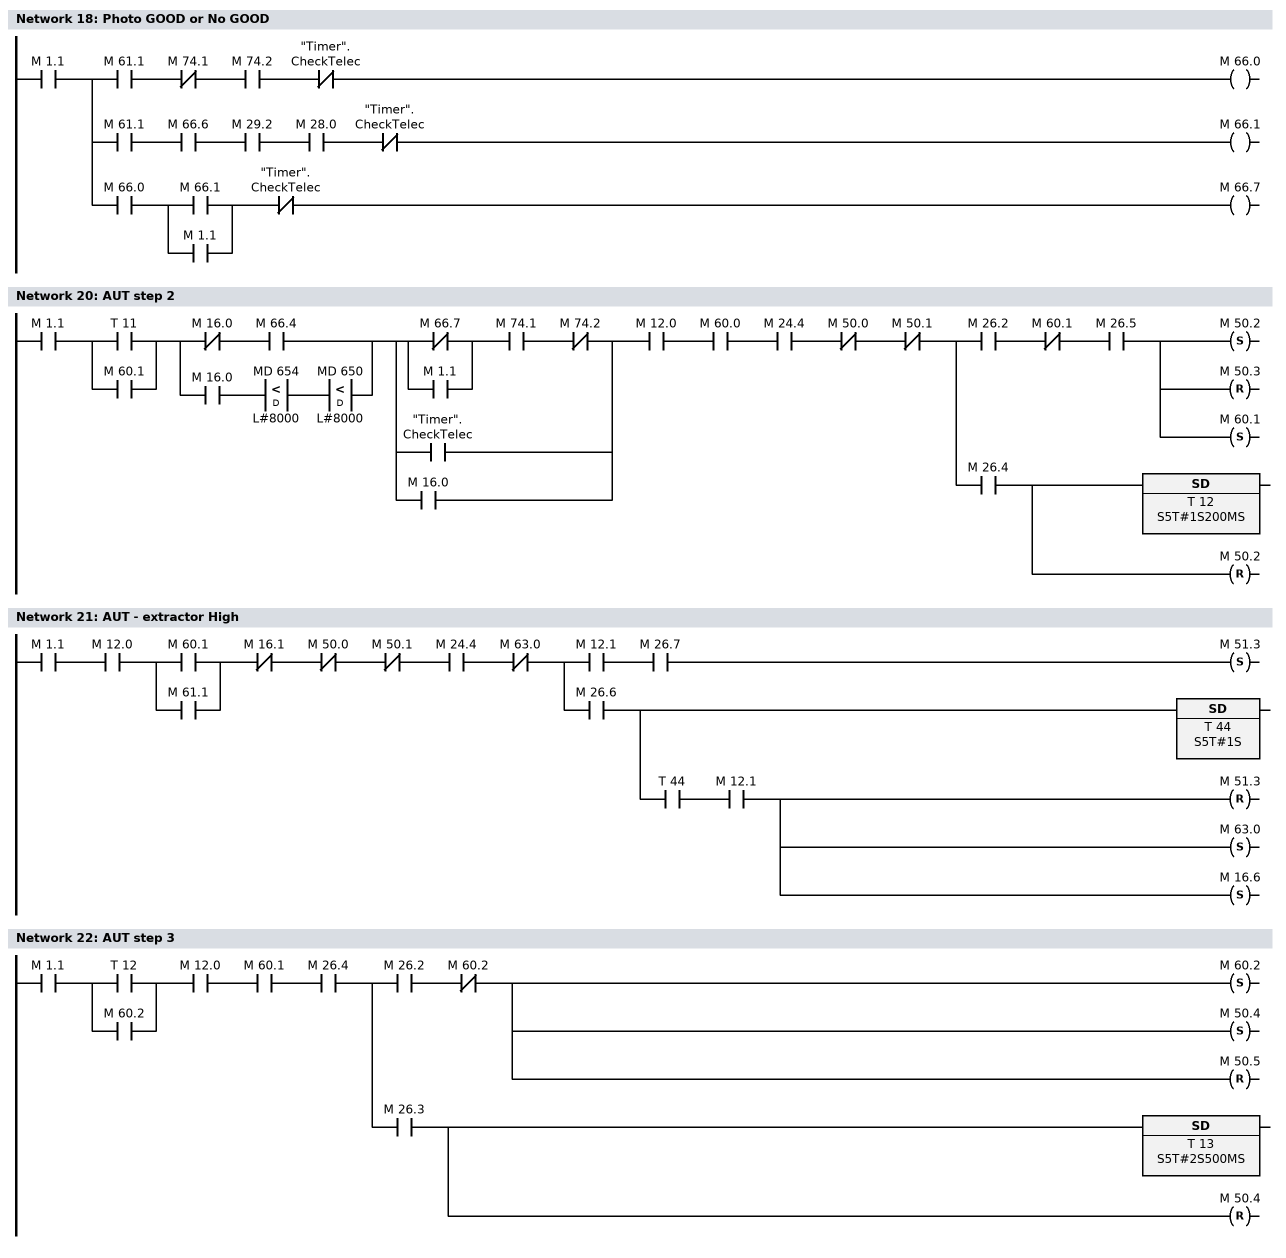
NETWORK
TITLE = Photo GOOD or No GOOD
      A     M 1.1;
      =     L 16.0;
      A     L 16.0;
      A     M 61.1;
      AN    M 74.1;
      A     M 74.2;
      AN    "Timer".CheckTelec;
      =     M 66.0;
      A     L 16.0;
      A     M 61.1;
      A     M 66.6;
      A     M 29.2;
      A     M 28.0;
      AN    "Timer".CheckTelec;
      =     M 66.1;
      A     L 16.0;
      A     M 66.0;
      A(;
      O     M 66.1;
      O     M 1.1;
      );
      AN    "Timer".CheckTelec;
      =     M 66.7;
NETWORK
TITLE =
NETWORK
TITLE = AUT step 2
//Step 2: System Detector Forward ed 
      A     M 1.1;
      A(;
      O     T 11;
      O     M 60.1;
      );
      A(;
      AN    M 16.0;
      A     M 66.4;
      O;
      A     M 16.0;
      A(;
      L     MD 654;
      L     L#8000;
      <D;
      );
      A(;
      L     MD 650;
      L     L#8000;
      <D;
      );
      );
      A(;
      A(;
      ON    M 66.7;
      O     M 1.1;
      );
      A     M 74.1;
      AN    M 74.2;
      O     "Timer".CheckTelec;
      O     M 16.0;
      );
      A     M 12.0;
      A     M 60.0;
      A     M 24.4;
      AN    M 50.0;
      AN    M 50.1;
      =     L 16.0;
      A     L 16.0;
      A     M 26.2;
      AN    M 60.1;
      A     M 26.5;
      S     M 50.2;
      R     M 50.3;
      S     M 60.1;
      A     L 16.0;
      A     M 26.4;
      L     S5T#1S200MS;
      SD    T 12;
      R     M 50.2;
NETWORK
TITLE = AUT - extractor High
//Insert Extractor , extract worked pieces, i make it together Step 2
      A     M 1.1;
      A     M 12.0;
      A(;
      O     M 60.1;
      O     M 61.1;
      );
      AN    M 16.1;
      AN    M 50.0;
      AN    M 50.1;
      A     M 24.4;
      AN    M 63.0;
      =     L 16.0;
      A     L 16.0;
      A     M 12.1;
      A     M 26.7;
      S     M 51.3;
      A     L 16.0;
      A     M 26.6;
      =     L 16.1;
      A     L 16.1;
      BLD   102;
      L     S5T#1S;
      SD    T 44;
      A     L 16.1;
      A     T 44;
      A     M 12.1;
      R     M 51.3;
      S     M 63.0;
      S     M 16.6;
NETWORK
TITLE = AUT step 3
//Step 3: System Detector Low
      A     M 1.1;
      A(;
      O     T 12;
      O     M 60.2;
      );
      A     M 12.0;
      A     M 60.1;
      A     M 26.4;
      =     L 16.0;
      A     L 16.0;
      A     M 26.2;
      AN    M 60.2;
      S     M 60.2;
      S     M 50.4;
      R     M 50.5;
      A     L 16.0;
      A     M 26.3;
      L     S5T#2S500MS;
      SD    T 13;
      R     M 50.4;
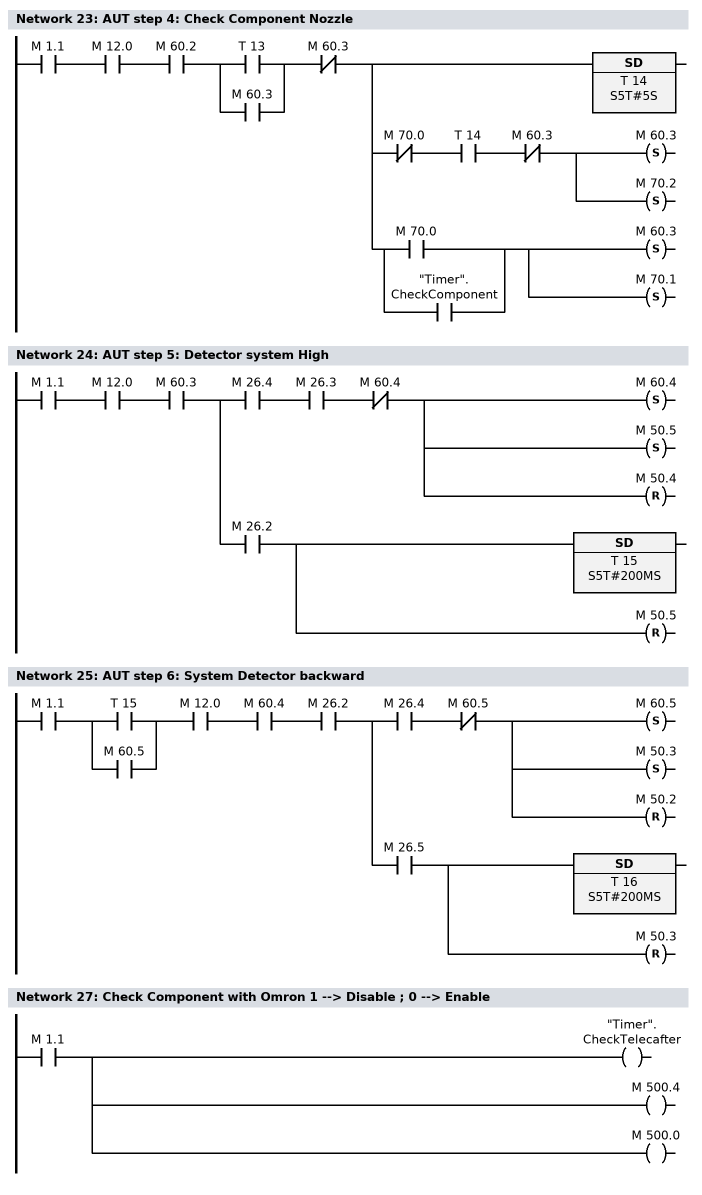
NETWORK
TITLE = AUT step 4: Check Component Nozzle
//check if is possible work pieces
//
      A     M 1.1;
      A     M 12.0;
      A     M 60.2;
      A(;
      O     T 13;
      O     M 60.3;
      );
      AN    M 60.3;
      =     L 16.0;
      A     L 16.0;
      BLD   102;
      L     S5T#5S;
      SD    T 14;
      A     L 16.0;
      AN    M 70.0;
      A     T 14;
      AN    M 60.3;
      S     M 60.3;
      S     M 70.2;
      A     L 16.0;
      A(;
      O     M 70.0;
      O     "Timer".CheckComponent;
      );
      S     M 60.3;
      S     M 70.1;
NETWORK
TITLE = AUT step 5: Detector system High
      A     M 1.1;
      A     M 12.0;
      A     M 60.3;
      =     L 16.0;
      A     L 16.0;
      A     M 26.4;
      A     M 26.3;
      AN    M 60.4;
      S     M 60.4;
      S     M 50.5;
      R     M 50.4;
      A     L 16.0;
      A     M 26.2;
      L     S5T#200MS;
      SD    T 15;
      R     M 50.5;
NETWORK
TITLE = AUT step 6: System Detector backward
//torno con il controllo in posizione iniziale
      A     M 1.1;
      A(;
      O     T 15;
      O     M 60.5;
      );
      A     M 12.0;
      A     M 60.4;
      A     M 26.2;
      =     L 16.0;
      A     L 16.0;
      A     M 26.4;
      AN    M 60.5;
      S     M 60.5;
      S     M 50.3;
      R     M 50.2;
      A     L 16.0;
      A     M 26.5;
      L     S5T#200MS;
      SD    T 16;
      R     M 50.3;
NETWORK
TITLE =
NETWORK
TITLE = Check Component with Omron 1 --> Disable ; 0 --> Enable
      A     M 1.1;
      =     "Timer".CheckTelecafter;
      =     M 500.4;
      =     M 500.0;
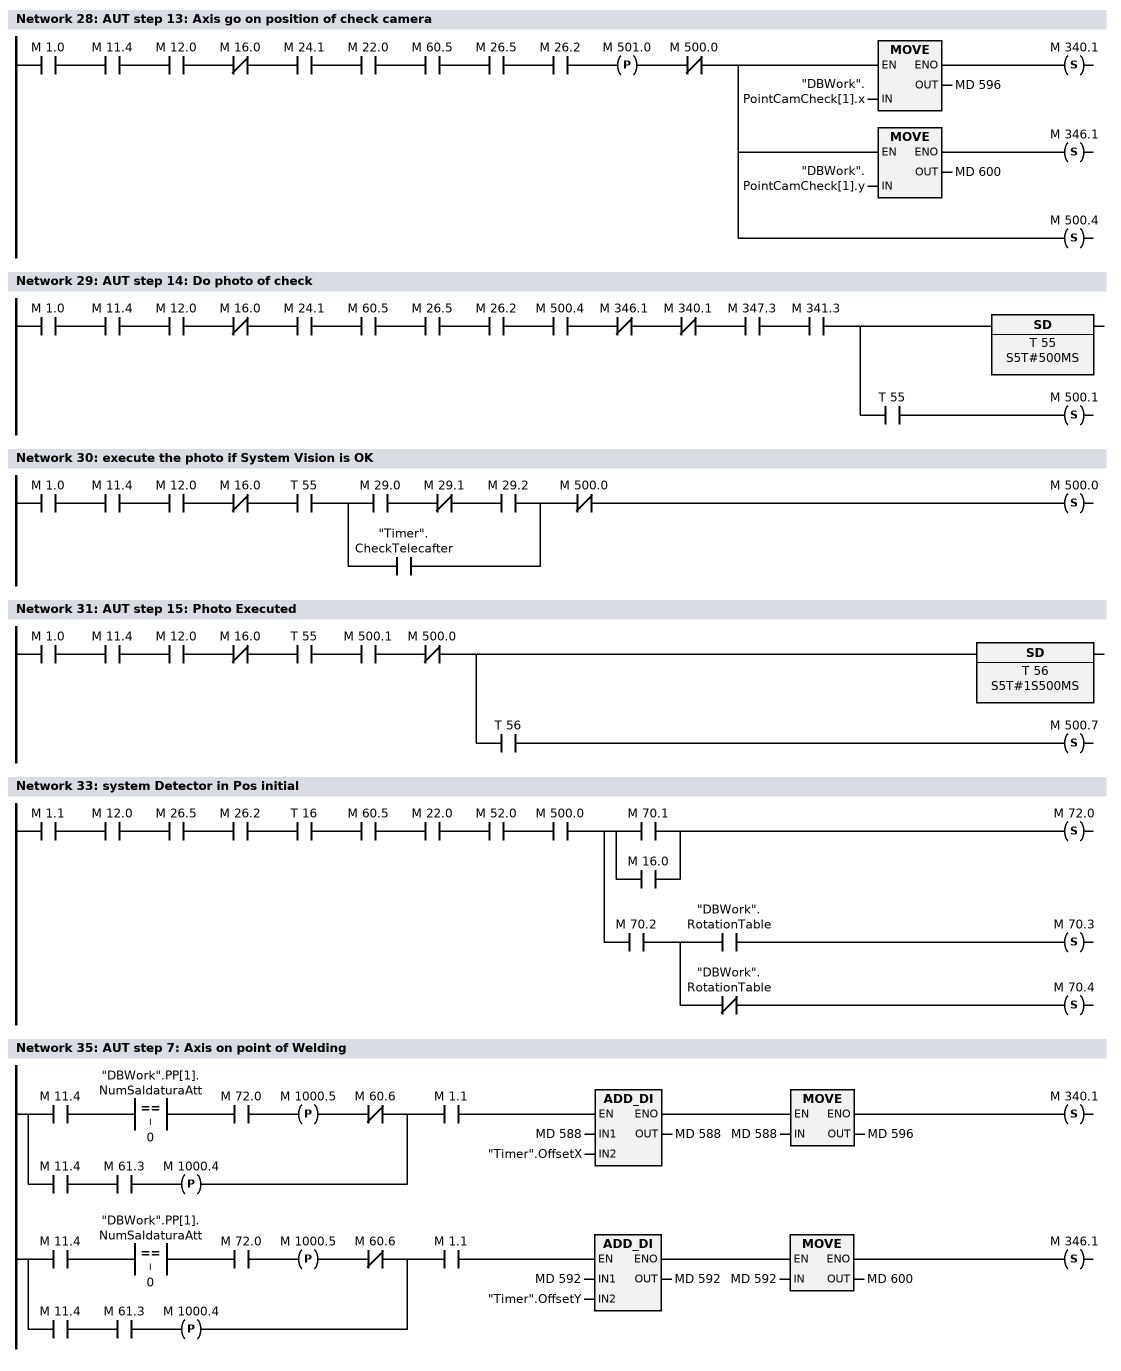
NETWORK
TITLE = AUT step 13: Axis go on position of check camera
      A     M 1.0;
      A     M 11.4;
      A     M 12.0;
      AN    M 16.0;
      A     M 24.1;
      A     M 22.0;
      A     M 60.5;
      A     M 26.5;
      A     M 26.2;
      FP    M 501.0;
      AN    M 500.0;
      =     L 16.0;
      A     L 16.0;
      JNB   _008;
      L     "DBWork".PointCamCheck[1].x;
      T     MD 596;
      SET;
      SAVE;
      CLR;
_008: A     BR;
      S     M 340.1;
      A     L 16.0;
      JNB   _009;
      L     "DBWork".PointCamCheck[1].y;
      T     MD 600;
      SET;
      SAVE;
      CLR;
_009: A     BR;
      S     M 346.1;
      A     L 16.0;
      BLD   102;
      S     M 500.4;
NETWORK
TITLE = AUT step 14: Do photo of check 
      A     M 1.0;
      A     M 11.4;
      A     M 12.0;
      AN    M 16.0;
      A     M 24.1;
      A     M 60.5;
      A     M 26.5;
      A     M 26.2;
      A     M 500.4;
      AN    M 346.1;
      AN    M 340.1;
      A     M 347.3;
      A     M 341.3;
      =     L 16.0;
      A     L 16.0;
      BLD   102;
      L     S5T#500MS;
      SD    T 55;
      A     L 16.0;
      A     T 55;
      S     M 500.1;
NETWORK
TITLE = execute the photo if System Vision is OK
      A     M 1.0;
      A     M 11.4;
      A     M 12.0;
      AN    M 16.0;
      A     T 55;
      A(;
      A     M 29.0;
      AN    M 29.1;
      A     M 29.2;
      O     "Timer".CheckTelecafter;
      );
      AN    M 500.0;
      S     M 500.0;
NETWORK
TITLE = AUT step 15: Photo Executed
      A     M 1.0;
      A     M 11.4;
      A     M 12.0;
      AN    M 16.0;
      A     T 55;
      A     M 500.1;
      AN    M 500.0;
      =     L 16.0;
      A     L 16.0;
      BLD   102;
      L     S5T#1S500MS;
      SD    T 56;
      A     L 16.0;
      A     T 56;
      S     M 500.7;
NETWORK
TITLE =
NETWORK
TITLE = system Detector in Pos initial
//System Detector in Pos initial and ready for detect Welding point
      A     M 1.1;
      A     M 12.0;
      A     M 26.5;
      A     M 26.2;
      A     T 16;
      A     M 60.5;
      A     M 22.0;
      A     M 52.0;
      A     M 500.0;
      =     L 16.0;
      A     L 16.0;
      A(;
      O     M 70.1;
      O     M 16.0;
      );
      S     M 72.0;
      A     L 16.0;
      A     M 70.2;
      =     L 16.1;
      A     L 16.1;
      A     "DBWork".RotationTable;
      S     M 70.3;
      A     L 16.1;
      AN    "DBWork".RotationTable;
      S     M 70.4;
NETWORK
TITLE = ------------START WITH WELDING
NETWORK
TITLE = AUT step 7: Axis on point of Welding
//AXIS X 
//AXIS Y 
//
//MD588 = SUPPORT FOR POINT X
//MD592 = SUPPORT FOR POINT Y
      A(;
      A     M 11.4;
      A(;
      L     "DBWork".PP[1].NumSaldaturaAtt;
      L     0;
      ==I;
      );
      A     M 72.0;
      FP    M 1000.5;
      AN    M 60.6;
      O(;
      A     M 11.4;
      A     M 61.3;
      FP    M 1000.4;
      );
      );
      A     M 1.1;
      =     L 16.0;
      A(;
      A     L 16.0;
      JNB   _00a;
      L     MD 588;
      L     "Timer".OffsetX;
      +D;
      T     MD 588;
      AN    OV;
      SAVE;
      CLR;
_00a: A     BR;
      );
      JNB   _00b;
      L     MD 588;
      T     MD 596;
      SET;
      SAVE;
      CLR;
_00b: A     BR;
      S     M 340.1;
      A(;
      A     L 16.0;
      JNB   _00c;
      L     MD 592;
      L     "Timer".OffsetY;
      +D;
      T     MD 592;
      AN    OV;
      SAVE;
      CLR;
_00c: A     BR;
      );
      JNB   _00d;
      L     MD 592;
      T     MD 600;
      SET;
      SAVE;
      CLR;
_00d: A     BR;
      S     M 346.1;
